// TwinCAT 3 PLC project Untitled1
// ProgramVersion: 3.1.4024.0
// libraries:
//   Tc2_Math, * (Beckhoff Automation GmbH)
//   Tc2_MC2, * (Beckhoff Automation GmbH)
//   Tc2_Standard, * (Beckhoff Automation GmbH)
//   Tc2_System, * (Beckhoff Automation GmbH)
//   Tc2_Utilities, * (Beckhoff Automation GmbH)
//   Tc3_Module, * (Beckhoff Automation GmbH)
//   Tc3_PackML_V2, * (Beckhoff Automation GmbH)
// project tree:
//   DUTs/DUTs/ E_ActWorkUnits.TcDUT (not stored), E_PMLUserUnitMode.TcDUT, E_UnitName.TcDUT (not stored), E_UnitTask.TcDUT (not stored), ST_FeedPara.TcDUT, ST_AxFunctions_1.TcDUT (not stored), ST_AxFunctionsAdmin_.TcDUT, ST_AxFunctionsPTP_1.TcDUT (not stored), ST_ChangeIntoProduction_1.TcDUT, ST_Folder.TcDUT (not stored), ST_FolderCom.TcDUT (not stored), ST_FolderPara.TcDUT, ST_FolderStatus.TcDUT, ST_OneJob.TcDUT (not stored), ST_UnitInfo.TcDUT (not stored)
//   / GlobalTextList.TcGTLO, PlcTask.TcTTO, 视图管理器.TcVMO (not stored)
//   GVLs/ APP_Com.TcDUT, GVL.TcGVL, GVL_Com.TcGVL (not stored), GVL_CONST.TcGVL, GVL_IO.TcGVL
//   POUs/Actuators/ AIN_EL3004.TcPOU (not stored), ANALOG_OUT.TcPOU (not stored), OUTPUT.TcPOU (not stored), SensorikAbblasen.TcPOU
//   POUs/Actuators/Cylinder/ CYLINDER.TcPOU
//   POUs/Actuators/FreqConv/ EcFcCom.TcPOU, IOFcCom.TcPOU
//   POUs/Actuators/Motor/ IOMotor.TcPOU (not stored), IOMotor2Dir.TcPOU (not stored), IOMotorStarDelta.TcPOU
//   POUs/ Axis_PTPV3_CoE.TcPOU, Ax_HMI.TcPOU (not stored), ERROR_HDL.TcPOU (not stored), fbMachine.TcPOU (not stored), FB_Generic.TcPOU (not stored), FB_Visu.TcPOU (not stored), INPUT.TcPOU (not stored), MAIN.TcPOU
//   POUs/EventLogger/ EventStatistik.TcPOU (not stored), EventStatistikData.TcPOU (not stored), EventsWriteToLogbook.TcPOU (not stored)
//   POUs/EventLogger/ReadEvents/ ReadAdsEvents.TcPOU (not stored), READ_ADS_EVENT_DATA.TcDUT, READ_ADS_EVENT_HANDLEINFO.TcDUT (not stored), READ_ADS_EVENT_STREAM.TcDUT, READ_ADS_EVENT_STREAM_DATA_EX.TcDUT (not stored), READ_ADS_EVENT_STREAM_DATA_RAW.TcDUT
//   POUs/EventLogger/TriggerEvents/ EventClass10.TcPOU (not stored), EventClass25.TcPOU, EventClass50.TcPOU (not stored), EventCtrl.TcPOU
//   POUs/Lib/ FB_HydLinearRamp.TcPOU
//   POUs/Lib/EventLogger/TriggerEvents/ EventClass50.TcPOU (not stored), EventCtrl.TcPOU (not stored)
//   POUs/PTP/00_DATATYPE/ AX_JOB.TcPOU (not stored)
//   POUs/PTP/01_Base/ Ax_AdminCtrl.TcPOU (not stored), Ax_HomingCtrl.TcPOU (not stored), Ax_MotionCtrl.TcPOU
//   POUs/PTP/02_Options/Coupling/ Ax_Camming.TcPOU (not stored) (excluded from build), Ax_FlySawCtrl.TcPOU (not stored) (excluded from build), Ax_GearCtrl.TcPOU (not stored)
//   POUs/PTP/02_Options/Drive/ Ax_BrakeCopperIO.TcPOU (not stored)
//   POUs/PTP/02_Options/Drive/CanOpen/ Ax_CanOpenDriveEventCtrl.TcPOU
//   POUs/PTP/02_Options/Drive/Ethercat/ Ax_Ax5000DriveCtrl.TcPOU (not stored), Ax_EcDriveEventCtrl.TcPOU (not stored), Ax_EcMC2DriveCtrl.TcPOU
//   POUs/PTP/02_Options/Drive/Stepper/ Ax_StepperDriveEventCtrl.TcPOU
//   POUs/PTP/02_Options/ErrorNc/ Ax_ErrorNCEventCtrl.TcPOU, Ax_ErrorNCEventMsgCtrl.TcPOU (not stored)
//   POUs/PTP/02_Options/Parameter/ Ax_Para.TcPOU (not stored), AX_PARA_SET_ISTPOS.TcPOU
//   POUs/PTP/02_Options/TouchProbe/ Ax_TouchProbeCtrl.TcPOU
//   POUs/PTP/03_Utilities/ Ax_AutoFctCtrl.TcPOU (not stored), Ax_LoopingDistanceCtrl.TcPOU, Ax_StateUnitCtrl.TcPOU (not stored) (excluded from build), GetAxErrTxt.TcPOU (not stored), MMIN_TO_MMS.TcPOU, MMS_TO_MMIN.TcPOU (not stored), SetOvrVelo.TcPOU
//   POUs/PulseGenerator/ PulseCtrl.TcPOU, PulseGeneratorCtrl.TcPOU
//   POUs/SystemInfo/ SystemInfoCtrl.TcPOU, TaskInfoCtrl.TcPOU
//   POUs/UNIT/fb_Apron/ Analog_To_Angle.TcPOU (not stored), Analog_To_Slide.TcPOU, Angle_To_Analog.TcPOU, fb_Apron.TcPOU (not stored), FB_FoldAbsPos.TcPOU (not stored), FB_SlideAbsPos.TcPOU, Slide_To_Analog.TcPOU
//   POUs/UNIT/fb_BackGauge/ fb_BackGauge.TcPOU (not stored), FB_BGAbsPos.TcPOU, FB_FeedAbsPos.TcPOU (not stored), FB_TblAbsPos.TcPOU (not stored)
//   POUs/UNIT/fb_Clamp/ Anolog_To_Height.TcPOU, fb_Clamp.TcPOU (not stored), FB_ClampJog.TcPOU, FB_ClampLock.TcPOU, FB_ClampMove.TcPOU (not stored), FB_ClampUnlock.TcPOU (not stored), Height_To_Anology.TcPOU (not stored)
//   POUs/UNIT/fb_Slitter/ fb_Slitter.TcPOU (not stored), FB_SlitterAct.TcPOU
//   VISUs/VISUs/Templates/ VIS_TemplateCommand.TcVIS (not stored), VIS_TemplateKeys.TcVIS (not stored), VIS_TemplatePMLStateModel.TcVIS
//   VISUs/VISUs/ VIS_Main.TcVIS (not stored)
// real-time tasks:
//   TASK PlcTask: cycle T#10ms, priority 20, ADS port 350
// motion (NC):
//   TASK NC-Task 1 SAF: cycle T#2ms, priority 4, ADS port 501
//   TASK NC-Task 1 SVB: cycle T#10ms, priority 8, ADS port 511
//   AXIS Axis_T1 (id 1)
//     Dynamic: Acceleration=3740, Deceleration=3740, Jerk=8038.85
//     OtherSettings: AllowMotionCmdToSlave=true
//     encoder EncType=19
//       EncPara: ScaleFactorNumerator=7e-05, MaxCount=#xffffffff, ReferenceSystem=1
//         SoftEndMinControl: Enable=true, Range=-25
//         SoftEndMaxControl: Enable=true, Range=1210
//     drive DrvType=16
//       DrvPara: MaxCount=#xffffffff, DriveControlDWord=#x00020000
//         Analog: VeloReferenz=300, TorqueSetpointScale=10, ScaleFactorActTorque=0.1
//         TimeComp: TaskDelayCycles=1
//     controller CtrType=1
//       CtrPara: PriorControlFactor=1
//         PosDiffControl: Range=10
//         Observer: BandWidth=20
//   AXIS Axis_T2 (id 2)
//     Dynamic: Acceleration=3740, Deceleration=3740, Jerk=8038.85
//     OtherSettings: AllowMotionCmdToSlave=true
//     encoder EncType=19
//       EncPara: ScaleFactorNumerator=7e-05, MaxCount=#xffffffff, ReferenceSystem=1
//         SoftEndMinControl: Enable=true, Range=-25
//         SoftEndMaxControl: Enable=true, Range=1210
//     drive DrvType=16
//       DrvPara: MaxCount=#xffffffff, DriveControlDWord=#x00020000
//         Analog: VeloReferenz=300, TorqueSetpointScale=10, ScaleFactorActTorque=0.1
//         TimeComp: TaskDelayCycles=1
//     controller CtrType=1
//       CtrPara: PriorControlFactor=1
//         PosDiffControl: Range=10
//         Observer: BandWidth=20
//   AXIS Axis_T3 (id 3)
//     Dynamic: Acceleration=3740, Deceleration=3740, Jerk=8038.85
//     OtherSettings: AllowMotionCmdToSlave=true
//     encoder EncType=19
//       EncPara: ScaleFactorNumerator=7e-05, Inverse=true, MaxCount=#xffffffff, ReferenceSystem=1
//         SoftEndMinControl: Range=-25
//         SoftEndMaxControl: Enable=true, Range=1210
//     drive DrvType=16
//       DrvPara: Inverse=true, MaxCount=#xffffffff, DriveControlDWord=#x00020000
//         Analog: VeloReferenz=300, TorqueSetpointScale=10, ScaleFactorActTorque=0.1
//         TimeComp: TaskDelayCycles=1
//     controller CtrType=1
//       CtrPara: PriorControlFactor=1
//         PosDiffControl: Range=10
//         Observer: BandWidth=20
//   AXIS Axis_T4 (id 4)
//     Dynamic: Acceleration=3740, Deceleration=3740, Jerk=8038.85
//     OtherSettings: AllowMotionCmdToSlave=true
//     encoder EncType=19
//       EncPara: ScaleFactorNumerator=7e-05, MaxCount=#xffffffff, ReferenceSystem=1
//         SoftEndMinControl: Enable=true, Range=-25
//         SoftEndMaxControl: Enable=true, Range=1210
//     drive DrvType=16
//       DrvPara: MaxCount=#xffffffff, DriveControlDWord=#x00020000
//         Analog: VeloReferenz=300, TorqueSetpointScale=10, ScaleFactorActTorque=0.1
//         TimeComp: TaskDelayCycles=1
//     controller CtrType=1
//       CtrPara: PriorControlFactor=1
//         PosDiffControl: Range=10
//         Observer: BandWidth=20
//   AXIS Axis_Table (id 9)
//     Dynamic: Acceleration=1200, Deceleration=1200, Jerk=1440
//     PositionAreaControl: Range=200
//     OtherSettings: AllowMotionCmdToSlave=true
//     encoder EncType=19
//       EncPara: Inverse=true, MaxCount=#xffffffff, ReferenceSystem=1
//         SoftEndMinControl: Range=-10
//         SoftEndMaxControl: Enable=true, Range=800
//     drive DrvType=16
//       DrvPara: Inverse=true, MaxCount=#xffffffff, DriveControlDWord=#x00020000
//         Analog: VeloReferenz=300, TorqueSetpointScale=10, ScaleFactorActTorque=0.1
//         TimeComp: TaskDelayCycles=1
//     controller CtrType=1
//       CtrPara: PriorControlFactor=1
//         PosDiffControl: Range=100
//         Observer: BandWidth=20
//   AXIS Axis_Feed (id 5)
//     PositionAreaControl: Range=200
//     OtherSettings: AllowMotionCmdToSlave=true
//     encoder EncType=19
//       EncPara: ScaleFactorNumerator=0.00026, MaxCount=#xffffffff, ReferenceSystem=1
//         SoftEndMinControl: Enable=true, Range=-420
//         SoftEndMaxControl: Enable=true, Range=3900
//     drive DrvType=16
//       DrvPara: MaxCount=#xffffffff, DriveControlDWord=#x00020000
//         Analog: TorqueSetpointScale=10, ScaleFactorActTorque=0.1
//         TimeComp: TaskDelayCycles=1
//     controller CtrType=1
//       CtrPara: PriorControlFactor=1
//         PosDiffControl: Range=200
//         Observer: BandWidth=20
// I/O:
//   DEVICE Device 2 (EtherCAT), AmsNetId 192.168.78.10.3.1
//     Term 24 (EK1100) [EK1100 EtherCAT Coupler (2A E-Bus)]
//       Term 25 (EL1008) [EL1008 8Ch. Dig. Input 24V, 3ms]
//       Term 27 (EL1008) [EL1008 8Ch. Dig. Input 24V, 3ms]
//       Term 28 (EL1008) [EL1008 8Ch. Dig. Input 24V, 3ms]
//       Term 30 (EL1008) [EL1008 8Ch. Dig. Input 24V, 3ms]
//       Term 31 (EL1008) [EL1008 8Ch. Dig. Input 24V, 3ms]
//       Term 33 (EL2008) [EL2008 8Ch. Dig. Output 24V, 0.5A]
//       Term 34 (EL2008) [EL2008 8Ch. Dig. Output 24V, 0.5A]
//       Term 35 (EL2008) [EL2008 8Ch. Dig. Output 24V, 0.5A]
//       Term 36 (EL2008) [EL2008 8Ch. Dig. Output 24V, 0.5A]
//       Term 14 (EL2008) [EL2008 8Ch. Dig. Output 24V, 0.5A]
//       Term 37 (EL3004) [EL3004 4Ch. Ana. Input +/-10V]
//       Term 38 (EL3004) [EL3004 4Ch. Ana. Input +/-10V]
//       Term 39 (EL4004) [EL4004 4Ch. Ana. Output 0-10V, 12bit]
//       Term 41 (EL4024) [EL4024 4Ch. Ana. Output 4-20mA, 12bit]
//       Term 42 (EL4024) [EL4024 4Ch. Ana. Output 4-20mA, 12bit]
//       Term 43 (EL3024) [EL3024 4Ch. Ana. Input 4-20mA DIFF]
//       Term 47 (EL9011) [EL9011 End Terminal]
//     Drive 19 (ASDA-W3-E CoE Drive) [Delta ASDA-W3-E EtherCAT(CoE) Drive]
//       modules: Module 1 (W3 Servo Drive-Axis), Module 2 (W3 Servo Drive-Axis), Module 3 (W3 Servo Drive-Axis), Module 4 (W3 Servo Drive-Axis), Module 5 (W3 Servo Drive-Axis), Module 6 (W3 Servo Drive-Axis)
// variable links:
//   NC-Task 1 SAF/Axes/Axis_Feed <-> Device 2 (EtherCAT)/Drive 19 (ASDA-W3-E CoE Drive)
//     Drive/Inputs/In/nDataIn3[0] <-> Module 6 (W3 Servo Drive-Axis)/1st TxPDO Mapping/Actual Torque
//     Drive/Inputs/In/nDcOutputTime <-> InfoData/DcOutputShift
//     Drive/Inputs/In/nState1 <-> Module 6 (W3 Servo Drive-Axis)/1st TxPDO Mapping/Status Word
//     Drive/Inputs/In/nState2 <-> Module 6 (W3 Servo Drive-Axis)/1st TxPDO Mapping/Status Word @bit 8
//     Drive/Inputs/In/nState4 @bit 1 <-> WcState/InputToggle
//     Drive/Inputs/In/nState4 <-> WcState/WcState
//     Drive/Outputs/Out/nCtrl1 <-> Module 6 (W3 Servo Drive-Axis)/1st RxPDO Mapping/Control Word
//     Drive/Outputs/Out/nCtrl2 <-> Module 6 (W3 Servo Drive-Axis)/1st RxPDO Mapping/Control Word @bit 8
//     Drive/Outputs/Out/nDataOut1 <-> Module 6 (W3 Servo Drive-Axis)/1st RxPDO Mapping/TargetPosition
//     Drive/Outputs/Out/nDataOut2 <-> Module 6 (W3 Servo Drive-Axis)/1st RxPDO Mapping/TargetVelocity
//     Drive/Outputs/Out/nDataOut4[0] <-> Module 6 (W3 Servo Drive-Axis)/1st RxPDO Mapping/Target Torque
//     Enc/Inputs/In/nDataIn1 <-> Module 6 (W3 Servo Drive-Axis)/1st TxPDO Mapping/ActualPosition
//     Enc/Inputs/In/nDataIn3 <-> Module 6 (W3 Servo Drive-Axis)/1st TxPDO Mapping/Touch Probe Pos1 Pos Value
//     Enc/Inputs/In/nDataIn7 <-> Module 6 (W3 Servo Drive-Axis)/1st TxPDO Mapping/ActualVelocity
//     Enc/Inputs/In/nDcInputTime <-> InfoData/DcInputShift
//     Enc/Inputs/In/nState4 @bit 1 <-> WcState/InputToggle
//     Enc/Inputs/In/nState4 <-> WcState/WcState
//     Enc/Inputs/In/nState5 <-> Module 6 (W3 Servo Drive-Axis)/1st TxPDO Mapping/Touch Probe Status
//     Enc/Inputs/In/nState6 <-> Module 6 (W3 Servo Drive-Axis)/1st TxPDO Mapping/Touch Probe Status @bit 8
//     Enc/Outputs/Out/nCtrl5 <-> Module 6 (W3 Servo Drive-Axis)/1st RxPDO Mapping/Touch Probe Function
//     Enc/Outputs/Out/nCtrl6 <-> Module 6 (W3 Servo Drive-Axis)/1st RxPDO Mapping/Touch Probe Function @bit 8
//   NC-Task 1 SAF/Axes/Axis_T1 <-> Device 2 (EtherCAT)/Drive 19 (ASDA-W3-E CoE Drive)
//     Drive/Inputs/In/nDataIn3[0] <-> Module 1 (W3 Servo Drive-Axis)/1st TxPDO Mapping/Actual Torque
//     Drive/Inputs/In/nDcOutputTime <-> InfoData/DcOutputShift
//     Drive/Inputs/In/nState1 <-> Module 1 (W3 Servo Drive-Axis)/1st TxPDO Mapping/Status Word
//     Drive/Inputs/In/nState2 <-> Module 1 (W3 Servo Drive-Axis)/1st TxPDO Mapping/Status Word @bit 8
//     Drive/Inputs/In/nState4 @bit 1 <-> WcState/InputToggle
//     Drive/Inputs/In/nState4 <-> WcState/WcState
//     Drive/Outputs/Out/nCtrl1 <-> Module 1 (W3 Servo Drive-Axis)/1st RxPDO Mapping/Control Word
//     Drive/Outputs/Out/nCtrl2 <-> Module 1 (W3 Servo Drive-Axis)/1st RxPDO Mapping/Control Word @bit 8
//     Drive/Outputs/Out/nDataOut1 <-> Module 1 (W3 Servo Drive-Axis)/1st RxPDO Mapping/TargetPosition
//     Drive/Outputs/Out/nDataOut2 <-> Module 1 (W3 Servo Drive-Axis)/1st RxPDO Mapping/TargetVelocity
//     Drive/Outputs/Out/nDataOut4[0] <-> Module 1 (W3 Servo Drive-Axis)/1st RxPDO Mapping/Target Torque
//     Enc/Inputs/In/nDataIn1 <-> Module 1 (W3 Servo Drive-Axis)/1st TxPDO Mapping/ActualPosition
//     Enc/Inputs/In/nDataIn3 <-> Module 1 (W3 Servo Drive-Axis)/1st TxPDO Mapping/Touch Probe Pos1 Pos Value
//     Enc/Inputs/In/nDataIn7 <-> Module 1 (W3 Servo Drive-Axis)/1st TxPDO Mapping/ActualVelocity
//     Enc/Inputs/In/nDcInputTime <-> InfoData/DcInputShift
//     Enc/Inputs/In/nState4 @bit 1 <-> WcState/InputToggle
//     Enc/Inputs/In/nState4 <-> WcState/WcState
//     Enc/Inputs/In/nState5 <-> Module 1 (W3 Servo Drive-Axis)/1st TxPDO Mapping/Touch Probe Status
//     Enc/Inputs/In/nState6 <-> Module 1 (W3 Servo Drive-Axis)/1st TxPDO Mapping/Touch Probe Status @bit 8
//     Enc/Outputs/Out/nCtrl5 <-> Module 1 (W3 Servo Drive-Axis)/1st RxPDO Mapping/Touch Probe Function
//     Enc/Outputs/Out/nCtrl6 <-> Module 1 (W3 Servo Drive-Axis)/1st RxPDO Mapping/Touch Probe Function @bit 8
//   NC-Task 1 SAF/Axes/Axis_T2 <-> Device 2 (EtherCAT)/Drive 19 (ASDA-W3-E CoE Drive)
//     Drive/Inputs/In/nDataIn3[0] <-> Module 2 (W3 Servo Drive-Axis)/1st TxPDO Mapping/Actual Torque
//     Drive/Inputs/In/nDcOutputTime <-> InfoData/DcOutputShift
//     Drive/Inputs/In/nState1 <-> Module 2 (W3 Servo Drive-Axis)/1st TxPDO Mapping/Status Word
//     Drive/Inputs/In/nState2 <-> Module 2 (W3 Servo Drive-Axis)/1st TxPDO Mapping/Status Word @bit 8
//     Drive/Inputs/In/nState4 @bit 1 <-> WcState/InputToggle
//     Drive/Inputs/In/nState4 <-> WcState/WcState
//     Drive/Outputs/Out/nCtrl1 <-> Module 2 (W3 Servo Drive-Axis)/1st RxPDO Mapping/Control Word
//     Drive/Outputs/Out/nCtrl2 <-> Module 2 (W3 Servo Drive-Axis)/1st RxPDO Mapping/Control Word @bit 8
//     Drive/Outputs/Out/nDataOut1 <-> Module 2 (W3 Servo Drive-Axis)/1st RxPDO Mapping/TargetPosition
//     Drive/Outputs/Out/nDataOut2 <-> Module 2 (W3 Servo Drive-Axis)/1st RxPDO Mapping/TargetVelocity
//     Drive/Outputs/Out/nDataOut4[0] <-> Module 2 (W3 Servo Drive-Axis)/1st RxPDO Mapping/Target Torque
//     Enc/Inputs/In/nDataIn1 <-> Module 2 (W3 Servo Drive-Axis)/1st TxPDO Mapping/ActualPosition
//     Enc/Inputs/In/nDataIn3 <-> Module 2 (W3 Servo Drive-Axis)/1st TxPDO Mapping/Touch Probe Pos1 Pos Value
//     Enc/Inputs/In/nDataIn7 <-> Module 2 (W3 Servo Drive-Axis)/1st TxPDO Mapping/ActualVelocity
//     Enc/Inputs/In/nDcInputTime <-> InfoData/DcInputShift
//     Enc/Inputs/In/nState4 @bit 1 <-> WcState/InputToggle
//     Enc/Inputs/In/nState4 <-> WcState/WcState
//     Enc/Inputs/In/nState5 <-> Module 2 (W3 Servo Drive-Axis)/1st TxPDO Mapping/Touch Probe Status
//     Enc/Inputs/In/nState6 <-> Module 2 (W3 Servo Drive-Axis)/1st TxPDO Mapping/Touch Probe Status @bit 8
//     Enc/Outputs/Out/nCtrl5 <-> Module 2 (W3 Servo Drive-Axis)/1st RxPDO Mapping/Touch Probe Function
//     Enc/Outputs/Out/nCtrl6 <-> Module 2 (W3 Servo Drive-Axis)/1st RxPDO Mapping/Touch Probe Function @bit 8
//   NC-Task 1 SAF/Axes/Axis_T3 <-> Device 2 (EtherCAT)/Drive 19 (ASDA-W3-E CoE Drive)
//     Drive/Inputs/In/nDataIn3[0] <-> Module 3 (W3 Servo Drive-Axis)/1st TxPDO Mapping/Actual Torque
//     Drive/Inputs/In/nDcOutputTime <-> InfoData/DcOutputShift
//     Drive/Inputs/In/nState1 <-> Module 3 (W3 Servo Drive-Axis)/1st TxPDO Mapping/Status Word
//     Drive/Inputs/In/nState2 <-> Module 3 (W3 Servo Drive-Axis)/1st TxPDO Mapping/Status Word @bit 8
//     Drive/Inputs/In/nState4 @bit 1 <-> WcState/InputToggle
//     Drive/Inputs/In/nState4 <-> WcState/WcState
//     Drive/Outputs/Out/nCtrl1 <-> Module 3 (W3 Servo Drive-Axis)/1st RxPDO Mapping/Control Word
//     Drive/Outputs/Out/nCtrl2 <-> Module 3 (W3 Servo Drive-Axis)/1st RxPDO Mapping/Control Word @bit 8
//     Drive/Outputs/Out/nDataOut1 <-> Module 3 (W3 Servo Drive-Axis)/1st RxPDO Mapping/TargetPosition
//     Drive/Outputs/Out/nDataOut2 <-> Module 3 (W3 Servo Drive-Axis)/1st RxPDO Mapping/TargetVelocity
//     Drive/Outputs/Out/nDataOut4[0] <-> Module 3 (W3 Servo Drive-Axis)/1st RxPDO Mapping/Target Torque
//     Enc/Inputs/In/nDataIn1 <-> Module 3 (W3 Servo Drive-Axis)/1st TxPDO Mapping/ActualPosition
//     Enc/Inputs/In/nDataIn3 <-> Module 3 (W3 Servo Drive-Axis)/1st TxPDO Mapping/Touch Probe Pos1 Pos Value
//     Enc/Inputs/In/nDataIn7 <-> Module 3 (W3 Servo Drive-Axis)/1st TxPDO Mapping/ActualVelocity
//     Enc/Inputs/In/nDcInputTime <-> InfoData/DcInputShift
//     Enc/Inputs/In/nState4 @bit 1 <-> WcState/InputToggle
//     Enc/Inputs/In/nState4 <-> WcState/WcState
//     Enc/Inputs/In/nState5 <-> Module 3 (W3 Servo Drive-Axis)/1st TxPDO Mapping/Touch Probe Status
//     Enc/Inputs/In/nState6 <-> Module 3 (W3 Servo Drive-Axis)/1st TxPDO Mapping/Touch Probe Status @bit 8
//     Enc/Outputs/Out/nCtrl5 <-> Module 3 (W3 Servo Drive-Axis)/1st RxPDO Mapping/Touch Probe Function
//     Enc/Outputs/Out/nCtrl6 <-> Module 3 (W3 Servo Drive-Axis)/1st RxPDO Mapping/Touch Probe Function @bit 8
//   NC-Task 1 SAF/Axes/Axis_T4 <-> Device 2 (EtherCAT)/Drive 19 (ASDA-W3-E CoE Drive)
//     Drive/Inputs/In/nDataIn3[0] <-> Module 4 (W3 Servo Drive-Axis)/1st TxPDO Mapping/Actual Torque
//     Drive/Inputs/In/nDcOutputTime <-> InfoData/DcOutputShift
//     Drive/Inputs/In/nState1 <-> Module 4 (W3 Servo Drive-Axis)/1st TxPDO Mapping/Status Word
//     Drive/Inputs/In/nState2 <-> Module 4 (W3 Servo Drive-Axis)/1st TxPDO Mapping/Status Word @bit 8
//     Drive/Inputs/In/nState4 @bit 1 <-> WcState/InputToggle
//     Drive/Inputs/In/nState4 <-> WcState/WcState
//     Drive/Outputs/Out/nCtrl1 <-> Module 4 (W3 Servo Drive-Axis)/1st RxPDO Mapping/Control Word
//     Drive/Outputs/Out/nCtrl2 <-> Module 4 (W3 Servo Drive-Axis)/1st RxPDO Mapping/Control Word @bit 8
//     Drive/Outputs/Out/nDataOut1 <-> Module 4 (W3 Servo Drive-Axis)/1st RxPDO Mapping/TargetPosition
//     Drive/Outputs/Out/nDataOut2 <-> Module 4 (W3 Servo Drive-Axis)/1st RxPDO Mapping/TargetVelocity
//     Drive/Outputs/Out/nDataOut4[0] <-> Module 4 (W3 Servo Drive-Axis)/1st RxPDO Mapping/Target Torque
//     Enc/Inputs/In/nDataIn1 <-> Module 4 (W3 Servo Drive-Axis)/1st TxPDO Mapping/ActualPosition
//     Enc/Inputs/In/nDataIn3 <-> Module 4 (W3 Servo Drive-Axis)/1st TxPDO Mapping/Touch Probe Pos1 Pos Value
//     Enc/Inputs/In/nDataIn7 <-> Module 4 (W3 Servo Drive-Axis)/1st TxPDO Mapping/ActualVelocity
//     Enc/Inputs/In/nDcInputTime <-> InfoData/DcInputShift
//     Enc/Inputs/In/nState4 @bit 1 <-> WcState/InputToggle
//     Enc/Inputs/In/nState4 <-> WcState/WcState
//     Enc/Inputs/In/nState5 <-> Module 4 (W3 Servo Drive-Axis)/1st TxPDO Mapping/Touch Probe Status
//     Enc/Inputs/In/nState6 <-> Module 4 (W3 Servo Drive-Axis)/1st TxPDO Mapping/Touch Probe Status @bit 8
//     Enc/Outputs/Out/nCtrl5 <-> Module 4 (W3 Servo Drive-Axis)/1st RxPDO Mapping/Touch Probe Function
//     Enc/Outputs/Out/nCtrl6 <-> Module 4 (W3 Servo Drive-Axis)/1st RxPDO Mapping/Touch Probe Function @bit 8
//   NC-Task 1 SAF/Axes/Axis_Table <-> Device 2 (EtherCAT)/Drive 19 (ASDA-W3-E CoE Drive)
//     Drive/Inputs/In/nDataIn3[0] <-> Module 5 (W3 Servo Drive-Axis)/1st TxPDO Mapping/Actual Torque
//     Drive/Inputs/In/nDcOutputTime <-> InfoData/DcOutputShift
//     Drive/Inputs/In/nState1 <-> Module 5 (W3 Servo Drive-Axis)/1st TxPDO Mapping/Status Word
//     Drive/Inputs/In/nState2 <-> Module 5 (W3 Servo Drive-Axis)/1st TxPDO Mapping/Status Word @bit 8
//     Drive/Inputs/In/nState4 @bit 1 <-> WcState/InputToggle
//     Drive/Inputs/In/nState4 <-> WcState/WcState
//     Drive/Outputs/Out/nCtrl1 <-> Module 5 (W3 Servo Drive-Axis)/1st RxPDO Mapping/Control Word
//     Drive/Outputs/Out/nCtrl2 <-> Module 5 (W3 Servo Drive-Axis)/1st RxPDO Mapping/Control Word @bit 8
//     Drive/Outputs/Out/nDataOut1 <-> Module 5 (W3 Servo Drive-Axis)/1st RxPDO Mapping/TargetPosition
//     Drive/Outputs/Out/nDataOut2 <-> Module 5 (W3 Servo Drive-Axis)/1st RxPDO Mapping/TargetVelocity
//     Drive/Outputs/Out/nDataOut4[0] <-> Module 5 (W3 Servo Drive-Axis)/1st RxPDO Mapping/Target Torque
//     Enc/Inputs/In/nDataIn1 <-> Module 5 (W3 Servo Drive-Axis)/1st TxPDO Mapping/ActualPosition
//     Enc/Inputs/In/nDataIn3 <-> Module 5 (W3 Servo Drive-Axis)/1st TxPDO Mapping/Touch Probe Pos1 Pos Value
//     Enc/Inputs/In/nDataIn7 <-> Module 5 (W3 Servo Drive-Axis)/1st TxPDO Mapping/ActualVelocity
//     Enc/Inputs/In/nDcInputTime <-> InfoData/DcInputShift
//     Enc/Inputs/In/nState4 @bit 1 <-> WcState/InputToggle
//     Enc/Inputs/In/nState4 <-> WcState/WcState
//     Enc/Inputs/In/nState5 <-> Module 5 (W3 Servo Drive-Axis)/1st TxPDO Mapping/Touch Probe Status
//     Enc/Inputs/In/nState6 <-> Module 5 (W3 Servo Drive-Axis)/1st TxPDO Mapping/Touch Probe Status @bit 8
//     Enc/Outputs/Out/nCtrl5 <-> Module 5 (W3 Servo Drive-Axis)/1st RxPDO Mapping/Touch Probe Function
//     Enc/Outputs/Out/nCtrl6 <-> Module 5 (W3 Servo Drive-Axis)/1st RxPDO Mapping/Touch Probe Function @bit 8
//   Untitled1/Untitled1 Instance <-> Device 2 (EtherCAT)/Term 24 (EK1100)/Term 14 (EL2008)
//     PlcTask Outputs/GVL_IO.Out_EMG_RopeStop <-> Channel 8/Output
//     PlcTask Outputs/GVL_IO.Out_FlipCupSuction1 <-> Channel 2/Output
//     PlcTask Outputs/GVL_IO.Out_FlipCupSuction2 <-> Channel 4/Output
//     PlcTask Outputs/GVL_IO.Out_FlipCupVent1 <-> Channel 1/Output
//     PlcTask Outputs/GVL_IO.Out_FlipCupVent2 <-> Channel 3/Output
//     PlcTask Outputs/GVL_IO.Out_bak54 <-> Channel 5/Output
//     PlcTask Outputs/GVL_IO.Out_bak55 <-> Channel 6/Output
//     PlcTask Outputs/GVL_IO.Out_bak56 <-> Channel 7/Output
//   Untitled1/Untitled1 Instance <-> Device 2 (EtherCAT)/Term 24 (EK1100)/Term 25 (EL1008)
//     PlcTask Inputs/GVL_IO.In_btnReset <-> Channel 8/Input
//     PlcTask Inputs/GVL_IO.In_pedal1_Clamp <-> Channel 2/Input
//     PlcTask Inputs/GVL_IO.In_pedal1_Fold <-> Channel 5/Input
//     PlcTask Inputs/GVL_IO.In_pedal1_Gripper <-> Channel 6/Input
//     PlcTask Inputs/GVL_IO.In_pedal1_Slitter <-> Channel 3/Input
//     PlcTask Inputs/GVL_IO.In_pedal1_SlitterBack <-> Channel 4/Input
//     PlcTask Inputs/GVL_IO.In_pedal1_UnClamp <-> Channel 1/Input
//     PlcTask Inputs/GVL_IO.In_swOperator <-> Channel 7/Input
//   Untitled1/Untitled1 Instance <-> Device 2 (EtherCAT)/Term 24 (EK1100)/Term 27 (EL1008)
//     PlcTask Inputs/GVL_IO.In_sigBtmApron_FoldHome <-> Channel 7/Input
//     PlcTask Inputs/GVL_IO.In_sigBtmApron_SlideFWD <-> Channel 8/Input
//     PlcTask Inputs/GVL_IO.In_sigSlitLmt0 <-> Channel 1/Input
//     PlcTask Inputs/GVL_IO.In_sigSlitLmt1 <-> Channel 3/Input
//     PlcTask Inputs/GVL_IO.In_sigSlitSlw0 <-> Channel 2/Input
//     PlcTask Inputs/GVL_IO.In_sigSlitSlw1 <-> Channel 4/Input
//     PlcTask Inputs/GVL_IO.In_sigTopApron_FoldHome <-> Channel 5/Input
//     PlcTask Inputs/GVL_IO.In_sigTopApron_SlideFWD <-> Channel 6/Input
//   Untitled1/Untitled1 Instance <-> Device 2 (EtherCAT)/Term 24 (EK1100)/Term 28 (EL1008)
//     PlcTask Inputs/GVL_IO.In_SigSheetDetect1 <-> Channel 7/Input
//     PlcTask Inputs/GVL_IO.In_SigSheetDetect2 <-> Channel 8/Input
//     PlcTask Inputs/GVL_IO.In_bak35 <-> Channel 6/Input
//     PlcTask Inputs/GVL_IO.In_sigBoardPresent <-> Channel 5/Input
//     PlcTask Inputs/GVL_IO.In_sigClampMute <-> Channel 1/Input
//     PlcTask Inputs/GVL_IO.In_sigGaugingFrnt <-> Channel 2/Input
//     PlcTask Inputs/GVL_IO.In_sigGaugingMid <-> Channel 3/Input
//     PlcTask Inputs/GVL_IO.In_sigGaugingRear <-> Channel 4/Input
//   Untitled1/Untitled1 Instance <-> Device 2 (EtherCAT)/Term 24 (EK1100)/Term 30 (EL1008)
//     PlcTask Inputs/GVL_IO.In_EMG_RopeStop <-> Channel 6/Input
//     PlcTask Inputs/GVL_IO.In_sigLC_H <-> Channel 5/Input
//     PlcTask Inputs/GVL_IO.In_sigLC_VLong <-> Channel 4/Input
//     PlcTask Inputs/GVL_IO.In_sigLC_VShort <-> Channel 3/Input
//     PlcTask Inputs/GVL_IO.In_sigLaserFinger <-> Channel 2/Input
//     PlcTask Inputs/GVL_IO.In_sigLubeJam <-> Channel 8/Input
//     PlcTask Inputs/GVL_IO.In_sigPumpJam <-> Channel 7/Input
//     PlcTask Inputs/GVL_IO.In_swLC_Enable <-> Channel 1/Input
//   Untitled1/Untitled1 Instance <-> Device 2 (EtherCAT)/Term 24 (EK1100)/Term 31 (EL1008)
//     PlcTask Inputs/GVL_IO.In_EMG_HandleCabinet <-> Channel 2/Input
//     PlcTask Inputs/GVL_IO.In_EMG_MainCabinet <-> Channel 1/Input
//     PlcTask Inputs/GVL_IO.In_PowerON <-> Channel 3/Input
//     PlcTask Inputs/GVL_IO.In_PumpLow_Alarm <-> Channel 7/Input
//     PlcTask Inputs/GVL_IO.In_VltA_Running <-> Channel 4/Input
//     PlcTask Inputs/GVL_IO.In_VltB_Running <-> Channel 5/Input
//     PlcTask Inputs/GVL_IO.In_VltSlitter_Running <-> Channel 8/Input
//     PlcTask Inputs/GVL_IO.In_Vlt_Alarm <-> Channel 6/Input
//   Untitled1/Untitled1 Instance <-> Device 2 (EtherCAT)/Term 24 (EK1100)/Term 33 (EL2008)
//     PlcTask Outputs/GVL_IO.Out_ClampDown <-> Channel 2/Output
//     PlcTask Outputs/GVL_IO.Out_ClampUp <-> Channel 1/Output
//     PlcTask Outputs/GVL_IO.Out_PumpA_Load_Heav <-> Channel 6/Output
//     PlcTask Outputs/GVL_IO.Out_PumpA_Load_Ligh <-> Channel 5/Output
//     PlcTask Outputs/GVL_IO.Out_PumpB_Load_Heav <-> Channel 8/Output
//     PlcTask Outputs/GVL_IO.Out_PumpB_Load_Ligh <-> Channel 7/Output
//     PlcTask Outputs/GVL_IO.Out_SuctionCup1Suction <-> Channel 4/Output
//     PlcTask Outputs/GVL_IO.Out_SuctionCup1Vent <-> Channel 3/Output
//   Untitled1/Untitled1 Instance <-> Device 2 (EtherCAT)/Term 24 (EK1100)/Term 34 (EL2008)
//     PlcTask Outputs/GVL_IO.Out_GaugingF_Ext <-> Channel 1/Output
//     PlcTask Outputs/GVL_IO.Out_GaugingF_Rtn <-> Channel 2/Output
//     PlcTask Outputs/GVL_IO.Out_GaugingR_Ext <-> Channel 3/Output
//     PlcTask Outputs/GVL_IO.Out_GaugingR_Rtn <-> Channel 4/Output
//     PlcTask Outputs/GVL_IO.Out_Gripper <-> Channel 5/Output
//     PlcTask Outputs/GVL_IO.Out_Gripper2 <-> Channel 6/Output
//     PlcTask Outputs/GVL_IO.Out_GripperDatum_S0 <-> Channel 7/Output
//     PlcTask Outputs/GVL_IO.Out_GripperDatum_S1 <-> Channel 8/Output
//   Untitled1/Untitled1 Instance <-> Device 2 (EtherCAT)/Term 24 (EK1100)/Term 35 (EL2008)
//     PlcTask Outputs/GVL_IO.Out_LubePump <-> Channel 6/Output
//     PlcTask Outputs/GVL_IO.Out_PumpA_ST <-> Channel 1/Output
//     PlcTask Outputs/GVL_IO.Out_PumpB_ST <-> Channel 2/Output
//     PlcTask Outputs/GVL_IO.Out_SlitterBwd <-> Channel 4/Output
//     PlcTask Outputs/GVL_IO.Out_SlitterFwd <-> Channel 3/Output
//     PlcTask Outputs/GVL_IO.Out_SlitterSpeed <-> Channel 5/Output
//     PlcTask Outputs/GVL_IO.Out_SuctionCup2Suction <-> Channel 8/Output
//     PlcTask Outputs/GVL_IO.Out_SuctionCup2Vent <-> Channel 7/Output
//   Untitled1/Untitled1 Instance <-> Device 2 (EtherCAT)/Term 24 (EK1100)/Term 36 (EL2008)
//     PlcTask Outputs/GVL_IO.Out_Gripper3 <-> Channel 8/Output
//     PlcTask Outputs/GVL_IO.Out_Led_Green <-> Channel 7/Output
//     PlcTask Outputs/GVL_IO.Out_Led_Red <-> Channel 5/Output
//     PlcTask Outputs/GVL_IO.Out_Led_Yellow <-> Channel 6/Output
//     PlcTask Outputs/GVL_IO.Out_OpLed_Beep <-> Channel 4/Output
//     PlcTask Outputs/GVL_IO.Out_OpLed_Green <-> Channel 3/Output
//     PlcTask Outputs/GVL_IO.Out_OpLed_Red <-> Channel 1/Output
//     PlcTask Outputs/GVL_IO.Out_OpLed_Yellow <-> Channel 2/Output
//   Untitled1/Untitled1 Instance <-> Device 2 (EtherCAT)/Term 24 (EK1100)/Term 37 (EL3004)
//     PlcTask Inputs/GVL_IO.ANALOG_in_BtmApronFold <-> AI Standard Channel 3/Value
//     PlcTask Inputs/GVL_IO.ANALOG_in_BtmApronSlide <-> AI Standard Channel 4/Value
//     PlcTask Inputs/GVL_IO.ANALOG_in_TopApronFold <-> AI Standard Channel 1/Value
//     PlcTask Inputs/GVL_IO.ANALOG_in_TopApronSlide <-> AI Standard Channel 2/Value
//   Untitled1/Untitled1 Instance <-> Device 2 (EtherCAT)/Term 24 (EK1100)/Term 38 (EL3004)
//     PlcTask Inputs/GVL_IO.ANALOG_in_ClampHeight <-> AI Standard Channel 1/Value
//     PlcTask Inputs/GVL_IO.ANALOG_in_PumpPress <-> AI Standard Channel 2/Value
//     PlcTask Inputs/GVL_IO.ANALOG_in_bak23 <-> AI Standard Channel 3/Value
//     PlcTask Inputs/GVL_IO.ANALOG_in_bak24 <-> AI Standard Channel 4/Value
//   Untitled1/Untitled1 Instance <-> Device 2 (EtherCAT)/Term 24 (EK1100)/Term 39 (EL4004)
//     PlcTask Outputs/GVL_IO.ANALOG_out_PumpA <-> AO Outputs Channel 1/Analog output
//     PlcTask Outputs/GVL_IO.ANALOG_out_PumpB <-> AO Outputs Channel 2/Analog output
//     PlcTask Outputs/GVL_IO.ANALOG_out_bak3 <-> AO Outputs Channel 3/Analog output
//     PlcTask Outputs/GVL_IO.ANALOG_out_bak4 <-> AO Outputs Channel 4/Analog output
//   Untitled1/Untitled1 Instance <-> Device 2 (EtherCAT)/Term 24 (EK1100)/Term 41 (EL4024)
//     PlcTask Outputs/GVL_IO.ANALOG_out_BtmApronFold <-> AO Outputs Channel 1/Analog output
//     PlcTask Outputs/GVL_IO.ANALOG_out_BtmApronSlide <-> AO Outputs Channel 2/Analog output
//   Untitled1/Untitled1 Instance <-> Device 2 (EtherCAT)/Term 24 (EK1100)/Term 42 (EL4024)
//     PlcTask Outputs/GVL_IO.ANALOG_out_ClampDown <-> AO Outputs Channel 1/Analog output
//     PlcTask Outputs/GVL_IO.ANALOG_out_ClampUp <-> AO Outputs Channel 2/Analog output
//     PlcTask Outputs/GVL_IO.ANALOG_out_TopApronFold <-> AO Outputs Channel 3/Analog output
//     PlcTask Outputs/GVL_IO.ANALOG_out_TopApronSlide <-> AO Outputs Channel 4/Analog output
//   Untitled1/Untitled1 Instance <-> Device 2 (EtherCAT)/Term 24 (EK1100)/Term 43 (EL3024)
//     PlcTask Inputs/GVL_IO.ANALOG_in_LiquidHeight <-> AI Standard Channel 2/Value
//     PlcTask Inputs/GVL_IO.ANALOG_in_PumpTemp <-> AI Standard Channel 1/Value
//     PlcTask Inputs/GVL_IO.ANALOG_in_bak43 <-> AI Standard Channel 3/Value
//     PlcTask Inputs/GVL_IO.ANALOG_in_bak44 <-> AI Standard Channel 4/Value
//   Untitled1/Untitled1 Instance <-> NC-Task 1 SAF/Axes/Axis_Feed
//     PlcTask Inputs/MAIN.fbMachine.fbBackGauge.Axis_Feed.ref.NcToPlc <-> Outputs/ToPlc
//     PlcTask Outputs/MAIN.fbMachine.fbBackGauge.Axis_Feed.ref.PlcToNc <-> Inputs/FromPlc
//   Untitled1/Untitled1 Instance <-> NC-Task 1 SAF/Axes/Axis_T1
//     PlcTask Inputs/MAIN.fbMachine.fbBackGauge.Axis_T1.ref.NcToPlc <-> Outputs/ToPlc
//     PlcTask Outputs/MAIN.fbMachine.fbBackGauge.Axis_T1.ref.PlcToNc <-> Inputs/FromPlc
//   Untitled1/Untitled1 Instance <-> NC-Task 1 SAF/Axes/Axis_T2
//     PlcTask Inputs/MAIN.fbMachine.fbBackGauge.Axis_T2.ref.NcToPlc <-> Outputs/ToPlc
//     PlcTask Outputs/MAIN.fbMachine.fbBackGauge.Axis_T2.ref.PlcToNc <-> Inputs/FromPlc
//   Untitled1/Untitled1 Instance <-> NC-Task 1 SAF/Axes/Axis_T3
//     PlcTask Inputs/MAIN.fbMachine.fbBackGauge.Axis_T3.ref.NcToPlc <-> Outputs/ToPlc
//     PlcTask Outputs/MAIN.fbMachine.fbBackGauge.Axis_T3.ref.PlcToNc <-> Inputs/FromPlc
//   Untitled1/Untitled1 Instance <-> NC-Task 1 SAF/Axes/Axis_T4
//     PlcTask Inputs/MAIN.fbMachine.fbBackGauge.Axis_T4.ref.NcToPlc <-> Outputs/ToPlc
//     PlcTask Outputs/MAIN.fbMachine.fbBackGauge.Axis_T4.ref.PlcToNc <-> Inputs/FromPlc
//   Untitled1/Untitled1 Instance <-> NC-Task 1 SAF/Axes/Axis_Table
//     PlcTask Inputs/MAIN.fbMachine.fbBackGauge.Axis_Table.ref.NcToPlc <-> Outputs/ToPlc
//     PlcTask Outputs/MAIN.fbMachine.fbBackGauge.Axis_Table.ref.PlcToNc <-> Inputs/FromPlc

CONFIGURATION Untitled1
    RESOURCE PLC ON TwinCAT3
        TASK PlcTask(INTERVAL := T#10ms, PRIORITY := 20);
        PROGRAM MAIN WITH PlcTask : MAIN;
    END_RESOURCE
END_CONFIGURATION

// ---- DUTs/DUTs/E_PMLUserUnitMode.TcDUT
//Enumeration for User Modes
TYPE E_PMLUserUnitMode : (
	ePMLUnitMode_SemiAuto		:=  4,
	ePMLUnitMode_AutoSlitter	:=  5,
	ePMLUnitMode_Auto			:=  6,
	ePMLUnitMode_AutoFeed		:=  7,
	ePMLUnitMode_Usermode6 		:=  9,
	ePMLUnitMode_Usermode5 		:=  8,
	ePMLUnitMode_Usermode7 		:=  10
) DINT;
END_TYPE

// ---- DUTs/DUTs/ST_FeedPara.TcDUT
TYPE ST_FeedPara :
STRUCT
	Width:UINT;
	Length:UINT;
	Thickness:REAL;
	Quantity :UINT;
	Groups:UINT;
	Total:UINT;
	
	FeedPOS1:REAL;
	FeedPOS2:REAL;
	
END_STRUCT
END_TYPE

// ---- DUTs/DUTs/ST_AxFunctionsAdmin_.TcDUT
//structure includes axisfunctions
TYPE ST_AxFunctionsAdmin_ :
STRUCT
	Power	: MC_Power;
	Reset	: MC_Reset;
END_STRUCT
END_TYPE

// ---- DUTs/DUTs/ST_ChangeIntoProduction_1.TcDUT
//structure for a visu userwindow, to chnage into productionmode
TYPE ST_ChangeIntoProduction_1 :
STRUCT
	bYes		: BOOL;
	bNo			: BOOL;
	bYesReset	: BOOL;
END_STRUCT
END_TYPE

// ---- DUTs/DUTs/ST_FolderPara.TcDUT
TYPE ST_FolderPara :
STRUCT
	//[GlobalSwitch]
	swLightHeavy,swSimplexDuplex	:BOOL;
	swSlitterVelocity,swLoadingTable,swAngleDisplay	:BOOL;
	swLightCurtainEn	:BOOL;
	swClampOpen_InManual,swClampOpen_InAuto	:BOOL;
	swFeedMechanism:BOOL;
	// [ClampHeight]
	Clamp_LowPos,Clamp_MidPos,Clamp_HighPos	:REAL;
	Clamp_MaxPos,ClampHalfPos	:REAL;
	Clamp_PressFlat,Clamp_FoldEnd	:REAL;
	Clamp_FeedPos:REAL;
	// [BackgaugeApron]
	BackgaugeMaxPos,BackgaugeMinPos		:REAL;
	SlitterOffset	:REAL;			(*钳口－切刀的距离*)
	BtmApronZeroPosition,TopApronZeroPosition	:REAL;
	SquashBackstop_Top,SquashBackstop_Btm,SquashBackstop_External	:REAL;
	SquashBackstop_OpenTop,SquashBackstop_OpenBtm	:REAL;
	MT1_BackstopZero	:REAL;
	MT2_BackstopZero,MT3_BackstopZero,MT4_BackstopZero	:REAL;
	Flip_TableToClampDistance	:REAL;
	Flip_SuctionCupInstallPos	:REAL;
	Flip_PickupClampHeight		:REAL;
	Flip_TopApronPickupAngle	:REAL;
	Flip_TablePickupOffset		:REAL;
	//[ManualOldSelect]
	FoldMode,PosDatumPoint	:BOOL;
	SetFoldAngle,SetMoveBackgauge,SetTopApronSlide,SetBtmApronSlide,SetLoadingTable	:REAL;
	AngleAdditSel_id 		:REAL;

	
	bSemiAuto_Step,bSemiAuto_Slitter,bSemiAuto_BackGauge	:BOOL;
	//	[FEED]
	FeedOffset,FeedPosition	:REAL;
	SetMoveFeed	:REAL;
	
	BackGauge_MaxPos,	BackGauge_MinPos	:REAL;
	
	TopAngleAddit,BtmAngleAddit		:ARRAY[0..14] OF REAL;

END_STRUCT
END_TYPE

// ---- DUTs/DUTs/ST_FolderStatus.TcDUT
TYPE ST_FolderStatus :
STRUCT
	Mode	:INT;
	Operator	:INT;
	FoldRunning	:BOOL;
	Gripper,Gripper2	:BOOL;
	GripperClose,GripperHalf,GripperOpen :BOOL;

	SuctionCup1,SuctionCup2	:BOOL;	//真空吸盘
	FlipSuctionCup			:BOOL;	//翻转真空吸盘
	
	Slitter_AtHome	:BOOL;
	SlitterAtSlow	:BOOL;
	
	BackGauge_AtHome	:BOOL;
	BG_Coupled	:BOOL;
	
	ApronTopSlide_AtWork,ApronTopSlide_AtMax	:BOOL;
	ApronBtmSlide_AtWork,ApronBtmSlide_AtMax	:BOOL;
	ApronTopSlide_AtSlow,ApronBtmSlide_AtSlow	:BOOL;
	
	ApronTopFold_AtHome,ApronTopFold_AtMax		:BOOL;
	ApronBtmFold_AtHome,ApronBtmFold_AtMax		:BOOL;
	ApronFold_AtSlow	:BOOL;
	
	Clamp_AtPressPoint	:BOOL;
	Clamp_AtZeroPoint	:BOOL;
	Clamp_LtHalfPoint	:BOOL;
	Clamp_GtLowPoint	:BOOL;
	Clamp_Slow			:BOOL;
	
	Table_AtHome	:BOOL;
	
	Feed_AtHome	:BOOL;
	Feed_AtWork	:BOOL;
	
	Flip_WorkDone :BOOL;
	Flip_AtWork :BOOL;
END_STRUCT
END_TYPE

// ---- GVLs/APP_Com.TcDUT
TYPE APP_Com :
STRUCT
	bBackStationPosFinish:BOOL;
	bBendStationPosFinish:BOOL;
END_STRUCT
END_TYPE

// ---- POUs/EventLogger/ReadEvents/READ_ADS_EVENT_DATA.TcDUT
TYPE READ_ADS_EVENT_DATA :
STRUCT
	Class			: E_TcEventClass;
	id				: DWORD;
	State			: DWORD;
	Question		: DWORD;
	SourceId		: DWORD;
	Source			: STRING(80);
	DateAndTime		: DT;
	Computer		: STRING(80);
	MsgText			: STRING(500);
END_STRUCT
END_TYPE

// ---- POUs/EventLogger/ReadEvents/READ_ADS_EVENT_STREAM.TcDUT
TYPE READ_ADS_EVENT_STREAM :
STRUCT
	cbStream		: DWORD; 			(* size OF this structure, including all following TcGetEventParams structures *)
	count			: DWORD;
	data			: READ_ADS_EVENT_STREAM_DATA_RAW;	(* Stream OF TcGetEventParams *)
END_STRUCT
END_TYPE

// ---- POUs/EventLogger/ReadEvents/READ_ADS_EVENT_STREAM_DATA_RAW.TcDUT
TYPE READ_ADS_EVENT_STREAM_DATA_RAW :
STRUCT
	cb						: DWORD;
	InvokeId				: DWORD;
	Id						: DWORD;
	SrcId					: DWORD;
	addr					: ARRAY [1..8] OF BYTE;
	Class					: DWORD;
	Flags					: DWORD;
	Prio					: DWORD;
	State					: DWORD;
	UserData				: DWORD;
	zFmtProgId				: STRING(31);

	TimeSignaled			: T_FILETIME;
	TimeReset				: T_FILETIME;
	TimeConfirm				: T_FILETIME;

	evtData					: READ_ADS_EVENT_STREAM_DATA_EX;
	
END_STRUCT
END_TYPE

// ---- GVLs/GVL.TcGVL
VAR_GLOBAL
		PackTags					: ST_PackMLv30;					//PackTags
// Dekl. Global Taktmerker
	pulse													: PulseCtrl;

	// Dekl. GetSystemInfo
	SysInfo													: SystemInfoCtrl;
	
		bButtonProductionReq		: BOOL;							//TRUE when a mode change to PRODUCTION is requested
		
		
		aUnitInfo					: ARRAY [1..12] OF ST_UnitInfo;	//Array includes the states and modes of machineunits	
		aCaption					: ARRAY [1..12] OF STRING := ['F1','F2','F3','F4','F5','F6','F7','F8','F9','F10','F11','F12'];
		aKeyPressed					: ARRAY [1..12] OF BOOL;	
		
		//Axis1:AXIS_REF;
		
		SemiAuto_ActJob	:ST_OneJob;
		SemiAuto_LastJob , SemiAuto_NextJob	:ST_OneJob;
		SlitterAuto_ActJob_Width	:REAL;
		SlitterAuto_ActJob_Num	:REAL;
		FeedAuto_Job:ST_FeedPara;
		
	FirstDualPump_5m	:BOOL;
	
	bReset	:BOOL;
	rtReset	:R_TRIG;
	pedal_UnClamp,	pedal_Clamp		:BOOL;
	pedal_Slitter,	pedal_SlitterBack	:BOOL;
	pedal_Fold,	pedal_Gripper	:BOOL;

	
	Hmi_bArray		AT%MB0:ARRAY[0..299] OF BOOL;
	Hmi_iArray		AT%MW300:ARRAY[0..299] OF UINT;
	Hmi_rArray		AT%MD1000:ARRAY[0..299] OF REAL;
	
	
	
	Hmi_iSemiAuto 	AT%MW8000:ARRAY[0..299] OF INT;
	Hmi_iAuto 		AT%MW3000:ARRAY[0..299] OF INT;
	Hmi_rSlitter	AT%MW4000:ARRAY[0..29] OF REAL;
	
	
		
	stFolder		:ST_FOLDER;
	
	
	
	b_sigLC_VShort: BOOL;
	gvl_rtEnSemiAuto: R_trig;
	gvl_rtEnSlitter: R_trig;
	
	gvl_bSlipPatch_BtmSlide,gvl_bSlipPatch_BtmFold		:BOOL;

	
END_VAR



VAR_GLOBAL PERSISTENT
	i12345	:INT;
	b_SafeSysEn: BOOL;
	
	Operators	:UINT;
	LubePumpCount	:INT;
	
	stFolderPara	:ST_FolderPara;
	AngleMap_Top	AT%MW5000	:ARRAY[0..199] OF INT;
	AngleMap_Btm	AT%MW5500	:ARRAY[0..199] OF INT;
	HeightMap		AT%MW6000	:ARRAY[0..399] OF INT;
	AdvPara			AT%MW9000	:ARRAY[0..99]  OF REAL;
END_VAR


VAR_GLOBAL RETAIN
	gvl_rtEnManual: R_trig;
END_VAR

// ---- GVLs/GVL_CONST.TcGVL
VAR_GLOBAL CONSTANT
	PUMP_FREQ_IDLE: USINT  :=143;
	
	
	CONST_APRON_SLIDE_DECWINDOW			:REAL	:=30.0;				(*台板滑动减速距离*)
	CONST_APRON_SLIDE_WINDOW			:REAL	:=5.0;				(*台板滑动定位窗口*)
	CONST_APRON_TOPSLIDE_POS0		:REAL	:=0.0;			(*AtWork时为0*)
	CONST_APRON_TOPSLIDE_POS1		:REAL	:=50.0;
	CONST_APRON_TOPSLIDE_POS2		:REAL	:=100.0;
	CONST_APRON_TOPSLIDE_POS3		:REAL	:=195.0;		(*退回时为200*)

	CONST_APRON_BTMSLIDE_POS0		:REAL	:=0.0;			(*AtWork时为0*)
	CONST_APRON_BTMSLIDE_POS1		:REAL	:=50.0;
	CONST_APRON_BTMSLIDE_POS2		:REAL	:=100.0;
	CONST_APRON_BTMSLIDE_POS3		:REAL	:=195.0;		(*退回时为200*)

	
	CONST_APRON_FOLD_DECWINDOW			:REAL	:=10.0;				(*台板折弯减速距离*)
	CONST_APRON_FOLD_WINDOW				:REAL	:=20.0;				(*台板折弯定位窗口*)
	CONST_APRON_TOPFOLD_POS_MAX			:REAL	:=200.0;
	CONST_APRON_TOPFOLD_POS_MIN			:REAL	:=0.0;
	CONST_APRON_BTMFOLD_POS_Max			:REAL	:=200.0;
	CONST_APRON_BTMFOLD_POS_MIN			:REAL	:=0.0;
	CONST_APRON_TOPFOLD_LIMIT			:REAL	:=150.0;		(*上翻板折弯 -- 机械极限*)
	CONST_APRON_BTMFOLD_LIMIT			:REAL	:=150.0;		(*下翻板折弯 -- 机械极限*)
	
	CONST_CLAMP_LIGHT_PRESSURE_SETPOINT	:REAL	:=7.0;		(*钳口压紧的压力值*)	
	CONST_CLAMP_HEAVY_PRESSURE_SETPOINT	:INT	:=100;
	CONST_CLAMP_POS_CALIBRATION	:INT	:=4;		(*CLAMP calibration 定义为认为闭合的位置*)
	CONST_CLAMP_POS_HALF	:INT	:=45;
	CONST_CLAMP_POS_LOW	:INT	:=3;
	CONST_CLAMP_SPEED_CREEP	:INT	:=500;
	CONST_CLAMP_SPEED_HIGH	:INT	:=4000;
	CONST_CLAMP_MAXCONVERT		:DINT	:=10000;			(*模拟量为32767时对应的值*)
	
	CONST_BACKGAUGE_SPEED_HIGH	:INT	:=200;
	CONST_BACKGAUGE_SPEED_LOW	:INT	:=50;
	CONST_BACKGAUGE_SPEED_CREEP	:INT	:=20;
	CONST_BACKGAUGE_POS_ZERO	:INT	:=0;
	CONST_BACKGAUGE_POS_NegPlus	:INT	:=-20;
	CONST_BACKGAUGE_POS_Window	:REAL	:=2.0;
	
	CONST_BACKGAUGE_ATTACH_PUSH		:REAL	:=0.0;		(*附加量-PUSH*)
	CONST_BACKGAUGE_ATTACH_GRIP		:REAL	:=10.0;		(*附加量-GRIP*)
	CONST_BACKGAUGE_ATTACH_OVERGRIP	:REAL	:=30.0;		(*附加量-OVERGRIP*)
	CONST_BACKGAUGE_ATTACH_BACK		:REAL	:=60.0;		(*附加量-BACK*)
	
	CONST_TABLE_SPEED_HIGH	:INT	:=300;
	CONST_TABLE_POS_MAX		:INT	:=800;
	CONST_TABLE_POS_MIN		:INT	:=0;
	
	CONST_FEED_SPEED_HIGH	:INT	:=800;
	CONST_FEED_SPEED_LOW	:INT	:=500;
	CONST_FEED_SPEED_CREEP	:INT	:=20;
	CONST_FEED_POS_ZERO	:INT	:=0;
	CONST_FEED_POS_NegPlus	:INT	:=-20;
	CONST_FEED_POS_Window	:REAL	:=2.0;
	CONST_FEED_POS_MAX		:INT	:=3900;
	CONST_FEED_POS_MIN		:INT	:=-450;
	
END_VAR

VAR_GLOBAL 
	CNST_HYD_IDLE_SPD					:REAL	:=0.0;	//	油泵待机速度
	CNST_HYD_PUMP_ACC_STEP				:REAL	:=40.0;	//	油泵斜坡加速步长_初始值
	CNST_HYD_PUMP_DEC_STEP				:REAL	:=60.0;	//	油泵斜坡减速步长_初始值
	CNST_HYD_APRON_SLIDE_ACC_STEP		:REAL	:=80.0;	//	翻板滑动比例阀加速步长_初始值
	CNST_HYD_APRON_SLIDE_DEC_STEP		:REAL	:=120.0;	//	翻板滑动比例阀减速步长_初始值
	CNST_HYD_APRON_SLIDE_MIN_OUTPUT		:REAL	:=220.0;	//	翻板滑动比例阀最小起跳量_初始值
	CNST_HYD_APRON_FOLD_ACC_STEP		:REAL	:=70.0;	//	翻板折弯比例阀加速步长_初始值
	CNST_HYD_APRON_FOLD_DEC_STEP		:REAL	:=110.0;	//	翻板折弯比例阀减速步长_初始值
	CNST_HYD_APRON_FOLD_MIN_OUTPUT		:REAL	:=200.0;	//	翻板折弯比例阀最小起跳量_初始值
	CNST_HYD_CLAMP_ACC_STEP				:REAL	:=60.0;	//	夹钳比例阀加速步长_初始值
	CNST_HYD_CLAMP_DEC_STEP				:REAL	:=90.0;	//	夹钳比例阀减速步长_初始值
	CNST_HYD_CLAMP_MIN_OUTPUT			:REAL	:=180.0;	//	夹钳比例阀最小起跳量_初始值
							
	CNST_APRON_TOPSLIDE_FWD_SPD			:REAL	:=0.0;	//	上翻板滑动，前进，工作速度
	CNST_APRON_TOPSLIDE_FWD_CREEP_SPD	:REAL	:=0.0;	//	上翻板滑动，前进，爬行速度
	CNST_APRON_TOPSLIDE_BWD_SPD			:REAL	:=0.0;	//	上翻板滑动，后退，工作速度
	CNST_APRON_TOPSLIDE_BWD_CREEP_SPD	:REAL	:=0.0;	//	上翻板滑动，后退，爬行速度
								
	CNST_APRON_BTMSLIDE_FWD_SPD			:REAL	:=0.0;	//	下翻板滑动，前进，工作速度
	CNST_APRON_BTMSLIDE_FWD_CREEP_SPD	:REAL	:=0.0;	//	下翻板滑动，前进，爬行速度
	CNST_APRON_BTMSLIDE_BWD_SPD			:REAL	:=0.0;	//	下翻板滑动，后退，工作速度
	CNST_APRON_BTMSLIDE_BWD_CREEP_SPD	:REAL	:=0.0;	//	下翻板滑动，后退，爬行速度
							
	CNST_APRON_TOPSLIDE_FWD_DecDis		:REAL	:=0.0;	//	上翻板滑动，前进，减速距离
	CNST_APRON_TOPSLIDE_BWD_DecDis		:REAL	:=0.0;	//	上翻板滑动，后退，减速距离
	CNST_APRON_BTMSLIDE_FWD_DecDis		:REAL	:=0.0;	//	下翻板滑动，前进，减速距离
	CNST_APRON_BTMSLIDE_BWD_DecDis		:REAL	:=0.0;	//	下翻板滑动，后退，减速距离
	CNST_APRON_SLIDE_WINDOWS			:REAL	:=0.0;	//	翻板滑动，停止窗口
	CNST_APRON_TOPSLIDE_POS0			:REAL	:=0.0;	//	上翻板滑动，位置0
	CNST_APRON_TOPSLIDE_POS1			:REAL	:=0.0;	//	上翻板滑动，位置1
	CNST_APRON_TOPSLIDE_POS2			:REAL	:=0.0;	//	上翻板滑动，位置2
	CNST_APRON_TOPSLIDE_POS3			:REAL	:=0.0;	//	上翻板滑动，位置3
	CNST_APRON_BTMSLIDE_POS0			:REAL	:=0.0;	//	上翻板滑动，位置0
	CNST_APRON_BTMSLIDE_POS1			:REAL	:=0.0;	//	上翻板滑动，位置1
	CNST_APRON_BTMSLIDE_POS2			:REAL	:=0.0;	//	上翻板滑动，位置2
	CNST_APRON_BTMSLIDE_POS3			:REAL	:=0.0;	//	上翻板滑动，位置3
							
	CNST_APRON_TOPFOLD_FWD_SPD			:REAL	:=0.0;	//	上翻板折弯，前进，工作速度
	CNST_APRON_TOPFOLD_FWD_CREEP_SPD	:REAL	:=0.0;	//	上翻板折弯，前进，爬行速度
	CNST_APRON_TOPFOLD_BWD_SPD			:REAL	:=0.0;	//	上翻板折弯，后退，工作速度
	CNST_APRON_TOPFOLD_BWD_CREEP_SPD	:REAL	:=0.0;	//	上翻板折弯，后退，爬行速度
	CNST_APRON_BTMFOLD_FWD_SPD			:REAL	:=0.0;	//	下翻板折弯，前进，工作速度
	CNST_APRON_BTMFOLD_FWD_CREEP_SPD	:REAL	:=0.0;	//	下翻板折弯，前进，爬行速度
	CNST_APRON_BTMFOLD_BWD_SPD			:REAL	:=0.0;	//	下翻板折弯，后退，工作速度
	CNST_APRON_BTMFOLD_BWD_CREEP_SPD	:REAL	:=0.0;	//	下翻板折弯，后退，爬行速度
							
	CNST_APRON_TOPFOLD_FWD_DecDis_GT110	:REAL	:=0.0;	//	上翻板折弯，前进，>110度时，减速距离
	CNST_APRON_TOPFOLD_FWD_DecDis_LE110	:REAL	:=0.0;	//	上翻板折弯，后退，≤110度时，减速距离
	CNST_APRON_TOPFOLD_BWD_DecDis		:REAL	:=0.0;	//	上翻板折弯，后退，减速距离
	CNST_APRON_BTMFOLD_FWD_DecDis_GT110	:REAL	:=0.0;	//	下翻板折弯，前进，>110度时，减速距离
	CNST_APRON_BTMFOLD_FWD_DecDis_LE110	:REAL	:=0.0;	//	下翻板折弯，前进，≤110度时，减速距离
	CNST_APRON_BTMFOLD_BWD_DecDis		:REAL	:=0.0;	//	下翻板折弯，后退，减速距离
	CNST_APRON_FOLD_WINDOWS				:REAL	:=0.0;	//	翻板折弯，停止窗口
	CNST_APRON_TOPFOLD_MIN				:REAL	:=0.0;	//	上翻板折弯，最小极限
	CNST_APRON_TOPFOLD_MAX				:REAL	:=0.0;	//	上翻板折弯，最大极限
	CNST_APRON_BTMFOLD_MIN				:REAL	:=0.0;	//	下翻板折弯，最小极限
	CNST_APRON_BTMFOLD_MAX				:REAL	:=0.0;	//	下翻板折弯，最大极限
						
	CNST_CLAMP_OPEN_SPD_LT_HALF			:REAL	:=0.0;	//	钳口打开速度，低于半钳口位（手动模式）
	CNST_CLAMP_OPEN_SPD_GT_HALF			:REAL	:=0.0;	//	钳口打开速度，高于半钳口位
	CNST_CLAMP_CLOSE_SPD_LT_HALF		:REAL	:=0.0;	//	钳口下降速度，低于半钳口位
	CNST_CLAMP_CLOSE_SPD_GT_HALF		:REAL	:=0.0;	//	钳口下降速度，高于半钳口位
	CNST_CLAMP_LIGHT_PRESSURE_SETPOINT	:REAL	:=0.0;	//	钳口压紧时的压力值_轻型
	CNST_CLAMP_HEAVY_PRESSURE_SETPOINT	:REAL	:=0.0;	//	钳口压紧时的压力值_重型
	CNST_CLAMP_POS_CLOSED				:REAL	:=0.0;	//	钳口闭合位置
								
	CNST_BACKGAUGE_SPEED_HIGH			:REAL	:=0.0;	//	后夹送速度_高速
	CNST_BACKGAUGE_SPEED_LOW			:REAL	:=0.0;	//	后夹送速度_低速
	CNST_BACKGAUGE_ATTACH_PUSH			:REAL	:=0.0;	//	后夹送位置附加值_推动
	CNST_BACKGAUGE_ATTACH_GRIP			:REAL	:=0.0;	//	后夹送位置附加值_浅夹
	CNST_BACKGAUGE_ATTACH_OVERGRIP		:REAL	:=0.0;	//	后夹送位置附加值_深夹
	CNST_BACKGAUGE_ATTACH_BACK			:REAL	:=0.0;	//	后夹送位置附加值_后退
							
	CNST_TABLE_SPEED_HIGH				:REAL	:=0.0;	//	桌板速度_高速
	CNST_TABLE_POS_MAX					:REAL	:=0.0;	//	桌板限定位置_最大值
	CNST_TABLE_POS_MIN					:REAL	:=0.0;	//	桌板限定位置_最小值
								
	CNST_SLITTER_FWD_SPD				:REAL	:=0.0;	//	纵切前进，工作速度
	CNST_SLITTER_FWD_CREEP_SPD			:REAL	:=0.0;	//	纵切前进，爬行速度
	CNST_SLITTER_BWD_SPD				:REAL	:=0.0;	//	纵切后退，工作速度
	CNST_SLITTER_BWD_CREEP_SPD			:REAL	:=0.0;	//	纵切后退，爬行速度
								
	CNST_ANGLE_LIMIT_HEAVY				:REAL	:=0.0;	//	最大限制角度 重型
	CNST_ANGLE_LIMIT_LIGHT				:REAL	:=0.0;	//	最大限制角度 轻型
								
	CNST_LUBE_HYP_COUNTS				:REAL	:=0.0;	//	润滑泵注油动作计数
	CNST_LUBE_DURATION_WORK				:REAL	:=0.0;	//	润滑泵注油持续时间
	
	CNST_FEED_SPEED_HIGH				:INT	:=200;
	CNST_FEED_SPEED_LOW					:INT	:=50;
	CNST_FEED_SPEED_CREEP				:INT	:=20;
	CNST_FEED_POS_ZERO					:INT	:=0;
	CNST_FEED_POS_NegPlus				:INT	:=-20;
	CNST_FEED_POS_Window				:REAL	:=2.0;
	CNST_FEED_POS_MAX					:INT	:=5000;
	CNST_FEED_POS_MIN					:INT	:=-1000;
	
//	CNST_TAPER_REF_T1					:REAL	:=700.0;	//	锥度折弯 基准-T1距离
//	CNST_TAPER_REF_T2					:REAL	:=1460.0;	//	锥度折弯 基准-T2距离
//	CNST_TAPER_REF_T3					:REAL	:=2200.0;	//	锥度折弯 基准-T3距离
//	CNST_TAPER_REF_T4					:REAL	:=2960.0;	//	锥度折弯 基准-T4距离

	CNST_TAPER_REF						:REAL;
	CNST_TAPER_REF_T1					:REAL;
	CNST_TAPER_REF_T2					:REAL;
	CNST_TAPER_REF_T3					:REAL;
	CNST_TAPER_REF_T4					:REAL;

END_VAR

// ---- GVLs/GVL_IO.TcGVL

VAR_GLOBAL
(*------------------------------------------------Input Points-----------------------------------------*)
(*1st    EL1008  *)							
	In_pedal1_UnClamp		AT %I*		:BOOL;	(*脚踏1 -钳口放松*)
	In_pedal1_Clamp			AT %I*		:BOOL;	(*脚踏1 -钳口夹紧*)
	In_pedal1_Slitter		AT %I*		:BOOL;	(*脚踏1 -拉刀*)
	In_pedal1_SlitterBack	AT %I*		:BOOL;	(*脚踏1 -拉刀返回*)
	In_pedal1_Fold			AT %I*		:BOOL;	(*脚踏1 -折弯*)
	In_pedal1_Gripper		AT %I*		:BOOL;	(*脚踏1 -后定位夹钳*)
	In_swOperator			AT %I*		:BOOL;	(*操作员开/关*)
	In_btnReset				AT %I*		:BOOL;	(*复位*)
//(*2nd    EL1008  *)							
//	In_pedal_Autostart		AT %I*		:BOOL;	//开始折板	
//	In_bak11				AT %I*		:BOOL;	
//	In_bak12				AT %I*		:BOOL;	
//	In_bak13				AT %I*		:BOOL;	
//	In_bak14				AT %I*		:BOOL;	
//	In_bak15				AT %I*		:BOOL;	
//	In_bak16				AT %I*		:BOOL;	
//	In_bak17				AT %I*		:BOOL;	
(*3rd    EL1008  *)							
	In_sigSlitLmt0			AT %I*		:BOOL;	(*拉刀原点停止接近开关 *)
	In_sigSlitSlw0			AT %I*		:BOOL;	(*拉刀原点慢速接近开关*)
	In_sigSlitSlw1			AT %I*		:BOOL;	(*拉刀前进慢速接近开关*)
	In_sigSlitLmt1			AT %I*		:BOOL;	(*拉刀前进停止接近开关*)
	In_sigTopApron_FoldHome	AT %I*		:BOOL;	(*上翻板折弯原点接近开关*)
	In_sigTopApron_SlideFWD	AT %I*		:BOOL;	(*上翻板滑动前进接近开关*)
	In_sigBtmApron_FoldHome	AT %I*		:BOOL;	(*下翻板折弯原点接近开关*)
	In_sigBtmApron_SlideFWD	AT %I*		:BOOL;	(*下翻板滑动前进接近开关*)
(*4th    EL1008  *)							
	In_sigClampMute			AT %I*		:BOOL;	(*钳口静音接近开关 *)
	In_sigGaugingFrnt		AT %I*		:BOOL;	(*板厚接近开关1*)
	In_sigGaugingMid		AT %I*		:BOOL;	(*板厚接近开关2*)
	In_sigGaugingRear		AT %I*		:BOOL;	(*板厚接近开关3*)
	In_sigBoardPresent		AT %I*		:BOOL;	(*有板检测*)
	In_bak35				AT %I*		:BOOL;	(*备用2*)
	In_SigSheetDetect1		AT %I*		:BOOL;	(*板材检测1*)
	In_SigSheetDetect2		AT %I*		:BOOL;	(*板材检测2*)
//(*5th   EL1008  *)							
//	In_bak40				AT %I*		:BOOL;	
//	In_bak41				AT %I*		:BOOL;	
//	In_bak42				AT %I*		:BOOL;	
//	In_bak43				AT %I*		:BOOL;	
//	In_bak44				AT %I*		:BOOL;	
//	In_bak45				AT %I*		:BOOL;	
//	In_bak46				AT %I*		:BOOL;	
//	In_bak47				AT %I*		:BOOL;	
(*6th    EL1008  *)							
	In_swLC_Enable			AT %I*		:BOOL;	(*激光光幕校准开/关 *)
	In_sigLaserFinger		AT %I*		:BOOL;	(*激光传感器*)
	In_sigLC_VShort			AT %I*		:BOOL;	(*垂直光幕（短）*)
	In_sigLC_VLong			AT %I*		:BOOL;	(*垂直光幕（长）*)
	In_sigLC_H				AT %I*		:BOOL;	(*水平光幕*)
	In_EMG_RopeStop			AT %I*		:BOOL;	(*拉绳限位*)
	In_sigPumpJam			AT %I*		:BOOL;	(*油泵堵塞报警*)
	In_sigLubeJam			AT %I*		:BOOL;	(*润滑堵塞报警*)
(*7th    EL1008  *)							
	In_EMG_MainCabinet		AT %I*		:BOOL;	(*操作台急停*)
	In_EMG_HandleCabinet	AT %I*		:BOOL;	(*主控柜急停*)
	In_PowerON				AT %I*		:BOOL;	(*电源启动*)
	In_VltA_Running			AT %I*		:BOOL;	(*油泵变频A启动*)
	In_VltB_Running			AT %I*		:BOOL;	(*油泵变频B启动*)
	In_Vlt_Alarm			AT %I*		:BOOL;	(*变频无报警*)
	In_PumpLow_Alarm		AT %I*		:BOOL;	(*油泵液位低*)
	In_VltSlitter_Running	AT %I*		:BOOL;	(*拉刀变频启动*)

(*------------------------------------------------Output Points-----------------------------------------*)
(*1st    EL2008  *)
	Out_ApronBtm_SlideFWD	AT %Q*		:BOOL;	(*下翻板滑动前移*)
	Out_ApronBtm_SlideBWD	AT %Q*		:BOOL;	(*下翻板滑动后移*)
	Out_ApronBtm_FoldFWD	AT %Q*		:BOOL;	(*下翻板折弯前进*)
	Out_ApronBtm_FoldBWD	AT %Q*		:BOOL;	(*下翻板折弯返回*)
	Out_ApronTop_SlideFWD	AT %Q*		:BOOL;	(*上翻板滑动前移*)
	Out_ApronTop_SlideBWD	AT %Q*		:BOOL;	(*上翻板滑动后移*)
	Out_ApronTop_FoldFWD	AT %Q*		:BOOL;	(*上翻板折弯前进*)
	Out_ApronTop_FoldBWD	AT %Q*		:BOOL;	(*上翻板折弯返回*)
(*2nd    EL2008  *)							
	Out_ClampUp				AT %Q*		:BOOL;	(*钳口放松*)
	Out_ClampDown			AT %Q*		:BOOL;	(*钳口夹紧*)
	Out_SuctionCup1Vent		AT %Q*		:BOOL;	(*上料吸盘1放气*)
	Out_SuctionCup1Suction	AT %Q*		:BOOL;	(*上料吸盘1吸气*)
	Out_PumpB_Load_Ligh		AT %Q*		:BOOL;	(*泵B卸荷-轻型*)	
	Out_PumpB_Load_Heav		AT %Q*		:BOOL;	(*泵B卸荷-重型*)	
	Out_PumpA_Load_Ligh		AT %Q*		:BOOL;	(*泵A卸荷-轻型*)	
	Out_PumpA_Load_Heav		AT %Q*		:BOOL;	(*泵A卸荷-重型*)
(*3rd    EL2008  	Q2.x	*)
	Out_GaugingF_Ext		AT %Q*		:BOOL;	(*板厚调整油缸1伸出*)
	Out_GaugingF_Rtn		AT %Q*		:BOOL;	(*板厚调整油缸1缩回*)
	Out_GaugingR_Ext		AT %Q*		:BOOL;	(*板厚调整油缸2伸出*)
	Out_GaugingR_Rtn		AT %Q*		:BOOL;	(*板厚调整油缸2缩回*)
	Out_Gripper				AT %Q*		:BOOL;	(*后定位夹钳气缸夹紧*)
	Out_Gripper2			AT %Q*		:BOOL;	(*后定位夹钳气缸夹紧2*)
	Out_GripperDatum_S0		AT %Q*		:BOOL;	(*挡板气缸1伸出*)
	Out_GripperDatum_S1		AT %Q*		:BOOL;	(*挡板气缸2伸出*)
	(*
	Out_GripperDatum_S0  Out_GripperDatum_S1
       FALSE               FALSE           HOME
       TRUE                FALSE           PUSH
       FALSE               TRUE            GRIP
       TRUE                TRUE            OVERGRIP
	 *)
(*4th    EL2008  *)							
	Out_PumpA_ST			AT %Q*		:BOOL;	(*油泵A正转 *)
	Out_PumpB_ST			AT %Q*		:BOOL;	(*油泵B正转*)
	Out_SlitterFwd			AT %Q*		:BOOL;	(*拉刀正转*)
	Out_SlitterBwd			AT %Q*		:BOOL;	(*拉刀反转*)
	Out_SlitterSpeed		AT %Q*		:BOOL;	(*拉刀高低速*)
	Out_LubePump			AT %Q*		:BOOL;	(*润滑泵*)	
	Out_SuctionCup2Vent		AT %Q*		:BOOL;	(*上料吸盘2放气*)
	Out_SuctionCup2Suction	AT %Q*		:BOOL;	(*上料吸盘2吸气*)
(*5th    EL2008  *)							
	Out_OpLed_Red			AT %Q*		:BOOL;	(*操作员指示灯（红色）*)
	Out_OpLed_Yellow		AT %Q*		:BOOL;	(*操作员指示灯（黄色）*)	
	Out_OpLed_Green			AT %Q*		:BOOL;	(*操作员指示灯（绿色）*)
	Out_OpLed_Beep			AT %Q*		:BOOL;	(*操作员指示灯蜂鸣器*)
	Out_Led_Red				AT %Q*		:BOOL;	(*灯条(红色)*)	
	Out_Led_Yellow			AT %Q*		:BOOL;	(*灯条(黄色)*)
	Out_Led_Green			AT %Q*		:BOOL;	(*灯条(绿色)*)
	Out_Gripper3			AT %Q*		:BOOL;	(*后定位夹钳气缸夹紧3*)
(*6th    EL2008  *)							
	Out_FlipCupVent1		AT %Q*		:BOOL;	(*翻转吸盘放气*)
	Out_FlipCupSuction1		AT %Q*		:BOOL;	(*翻转吸盘吸气*)
	Out_FlipCupVent2		AT %Q*		:BOOL;	(*翻转吸盘放气*)
	Out_FlipCupSuction2		AT %Q*		:BOOL;	(*翻转吸盘吸气*)
	Out_bak54				AT %Q*		:BOOL;	(*备用*)
	Out_bak55				AT %Q*		:BOOL;	(*备用*)
	Out_bak56				AT %Q*		:BOOL;	(*备用*)
	Out_EMG_RopeStop		AT %Q*		:BOOL;	(*拉绳急停断电*)


	
(*------------------------------------------------ANALOG_in and out-----------------------------------------*)
	(*1th    EL3004  *)
	ANALOG_in_TopApronFold		AT %I*	:INT;	(*上翻板角度-位移传感器*)
	ANALOG_in_TopApronSlide		AT %I*	:INT;	(*上翻板滑动-位移传感器*)
	ANALOG_in_BtmApronFold		AT %I*	:INT;	(*下翻板角度-位移传感器*)
	ANALOG_in_BtmApronSlide		AT %I*	:INT;	(*下翻板滑动-位移传感器*)
	(*2th    EL3004  *)
	ANALOG_in_ClampHeight		AT %I*	:INT;	(*钳口高度    位移传感器*)
	ANALOG_in_PumpPress			AT %I*	:INT;	(*压力传感器*)
	ANALOG_in_bak23				AT %I*	:INT;	
	ANALOG_in_bak24				AT %I*	:INT;
	(*1th    EL4004  *)
	ANALOG_out_PumpA			AT %Q*	:INT;	(*油泵A调速*)
	ANALOG_out_PumpB			AT %Q*	:INT;	(*油泵B调速*)
	ANALOG_out_bak3				AT %Q*	:INT;
	ANALOG_out_bak4				AT %Q*	:INT;
	(*EL4024 4-20mA 比例阀输出*)
	ANALOG_out_BtmApronSlide	AT %Q*	:INT;	(*下翻板滑动比例阀 Term41 Ch2*)
	ANALOG_out_BtmApronFold		AT %Q*	:INT;	(*下翻板折弯比例阀 Term41 Ch1*)
	ANALOG_out_ClampUp			AT %Q*	:INT;	(*钳口放松比例阀 Term42 Ch2*)
	ANALOG_out_ClampDown		AT %Q*	:INT;	(*钳口夹紧比例阀 Term42 Ch1*)
	ANALOG_out_TopApronSlide	AT %Q*	:INT;	(*上翻板滑动比例阀 Term42 Ch4*)
	ANALOG_out_TopApronFold		AT %Q*	:INT;	(*上翻板折弯比例阀 Term42 Ch3*)
	(*1th    EL3024  *)
	ANALOG_in_PumpTemp			AT %I*	:INT;	(*油箱温度*)
	ANALOG_in_LiquidHeight		AT %I*	:INT;	(*液位高度*)
	ANALOG_in_bak43				AT %I*	:INT;	
	ANALOG_in_bak44				AT %I*	:INT;	
	
	(*Output AT %Q*: ARRAY [1..7, 1..8] OF BOOL;
	Input AT %I*: ARRAY [1..7, 1..8] OF BOOL;*)
END_VAR

// ---- POUs/MAIN.TcPOU
PROGRAM MAIN
VAR_EXTERNAL
	SysInfo													: SystemInfoCtrl;	 //Show online the global Sysinfo 
END_VAR
VAR
	TaskInfo												:	TaskInfoCtrl;
	bExecuteComplete			: BOOL;									//Command Execute Complete, not defined
	fbMachine:fbMachine;
	
	nStateCommandCheck: INT;
	
	fbVisu						: FB_Visu;		
	nCounter: INT;
	iBoot: INT;
	bBoot: BOOL;
	fbTon :TON;
	fbWritePersistentValue: WritePersistentData;
	i10 	:DINT;
	iModeSW: INT;
	ton1,ton2,ton3,ton4 :TON;
	B1: BOOL;
	i110: INT := 0;
	
	test1	:INPUT;
	test2: BOOL;
	rtTest2: R_trig;
	iAdd: INT;

END_VAR

TaskInfo();	
Boot();
ModeSw();

//Checking the Statecommands
CASE nStateCommandCheck OF
0:
	
	IF NOT FALSE THEN
		nStateCommandCheck:= 1;
	ELSE
		nStateCommandCheck:= 2;
	END_IF
	
1:
	IF PackTags.Command.CntrlCmd = ePMLCommand_Clear		
	  AND fbMachine.eState = ePMLState_Aborted	THEN
			fbMachine.eCommand	:= ePMLCommand_Clear;
	ELSIF PackTags.Command.CntrlCmd = ePMLCommand_Reset		
	  AND (fbMachine.eState = ePMLState_Stopped OR fbMachine.eState = ePMLState_Complete) THEN
			fbMachine.eCommand	:= ePMLCommand_Reset;
	ELSIF PackTags.Command.CntrlCmd = ePMLCommand_Start	
	  AND (fbMachine.eState = ePMLState_Idle OR (stPMLUnitModeConfiguration[fbMachine.eMode].aStateDisabled[ePMLState_Idle] AND fbMachine.eState = ePMLState_Stopped))
	  AND (NOT (PackTags.Command.Parameter[2].Value <= 0) OR NOT (fbMachine.eMode = 1))THEN
			fbMachine.eCommand	:= ePMLCommand_Start; 
	ELSIF PackTags.Command.CntrlCmd = ePMLCommand_Hold		
	  AND fbMachine.eState = ePMLState_Execute	
	  AND( fbMachine.eMode =  1 OR fbMachine.eMode =  4 OR fbMachine.eMode = 2)  THEN
			 fbMachine.eCommand	:= ePMLCommand_Hold;
	ELSIF PackTags.Command.CntrlCmd = ePMLCommand_Suspend	
	  AND fbMachine.eState = ePMLState_Execute	
	  AND (fbMachine.eMode = 4 OR fbMachine.eMode = 1)THEN
			 fbMachine.eCommand	:= ePMLCommand_Suspend;
	ELSIF PackTags.Command.CntrlCmd = ePMLCommand_Unhold	
	  AND fbMachine.eState = ePMLState_Held		THEN
			 fbMachine.eCommand	:= ePMLCommand_Unhold;
	ELSIF PackTags.Command.CntrlCmd = ePMLCommand_Unsuspend	
	  AND fbMachine.eState = ePMLState_Suspended	THEN
			 fbMachine.eCommand	:= ePMLCommand_Unsuspend;
	ELSIF PackTags.Command.CntrlCmd = ePMLCommand_Abort	THEN
			fbMachine.eCommand	:= ePMLCommand_Abort;
	ELSIF PackTags.Command.CntrlCmd = ePMLCommand_Stop	THEN
			fbMachine.eCommand	:= ePMLCommand_Stop;
	END_IF
	nStateCommandCheck:=0;
	
2:
	fbMachine.eCommand	:= ePMLCommand_Abort;
	IF fbMachine.eState = ePMLState_Aborted AND PackTags.Command.CntrlCmd = ePMLCommand_Clear THEN
		nStateCommandCheck:=1;
	END_IF
END_CASE

bButtonProductionReq := PackTags.Command.UnitMode = ePMLProtUnitMode_Production AND PackTags.Status.UnitModeCurrent <> PackTags.Command.UnitMode;

(*
fbMachine(
	eModeCommand:=PackTags.Command.UnitMode , 
	eCommand:=PackTags.Command.CntrlCmd , 
	eMode=>PackTags.Status.UnitModeCurrent , 
	eState=>PackTags.Status.StateCurrent , 
	bUndefinedDone=> , 
	bInvalidModeCommandOut=> , 
	bChangeIntoProduction=> );
	*)
fbMachine(eModeCommand:= PackTags.Command.UnitMode,  eMode => PackTags.Status.UnitModeCurrent, eState =>PackTags.Status.StateCurrent);
	
/// PackTags.Command.UnitModeChangeRequest;


  (* states according to PackTags v3.0 *)
  (*
    ePMLCommand_Undefined   := 0,
    ePMLCommand_Reset       := 1,
    ePMLCommand_Start       := 2,
    ePMLCommand_Stop        := 3,
    ePMLCommand_Hold        := 4,
    ePMLCommand_Unhold      := 5,
    ePMLCommand_Suspend     := 6,
    ePMLCommand_Unsuspend   := 7,
    ePMLCommand_Abort       := 8,
    ePMLCommand_Clear       := 9
	*)
	
M_Visu();

fbTon(IN:= NOT fbTon.Q , PT:=T#6S , Q=> , ET=> );
fbWritePersistentValue(
	NETID:='' ,
	PORT:= 851,
	START:=fbTon.Q ,
	TMOUT:=T#3s ,
	BUSY=> ,
	ERR=> ,
	ERRID=> );
IF fbTon.Q THEN
	i10:=i10+1;
END_IF;

(* Systemfunctions **********************************************************)
	SysInfo(
	RST:= , 
	RTCSyncCylce:=  , 
	TimeStampTrig:= pulse._100ms.RT , 
	ObjId=> , 
	TaskCnt=> , 
	OnlineChangeCount=> , 
	AppName=> , 
	AppTimestamp=> , 
	BootDataLoaded=> , 
	OldBootData=> , 
	TimeStampDT=> , 
	TimeStamp=> , 
	TimeStr=> , 
	DateStr=> , 
	TimeStamp2=> , 
	TimeStruct=> , 
	MonthDays=> , 
	LeapYear=> , 
	WeekOfYear=> , 
	timezoneId=> );

	Pulse();

	
	
	
	rtTest2(CLK:=Test2 , Q=> );
	test1(
	Force:= , 
	Invert:= , 
	PT_ON:=T#0S , 
	PT_OFF:=T#2S , 
	INPUT:=Test2 , 
	Q=> , 
	Q_RT=> , 
	Q_FT=> , 
	Q_DIRECT=> );

ACTION Boot:
(*
CASE iBoot OF
0:
iBoot	:=iBoot+1;
bBoot	:=TRUE;
1:	iBoot	:=iBoot+1;
2:	iBoot	:=iBoot+1;
3:	iBoot	:=iBoot+1;
4:	iBoot	:=iBoot+1;
5:
bBoot	:=FALSE;
RETURN;
END_CASE
*)
IF NOT TaskInfo.FirstCycle THEN
	RETURN;
END_IF

(*------------------------------------开机首次运行程序--------------------------*)
GVL.FirstDualPump_5m	:=TRUE;
Hmi_bArray[0]	:=stFolderPara.swSimplexDuplex;
Hmi_bArray[1]	:=stFolderPara.swLightHeavy;
Hmi_bArray[2]	:=stFolderPara.swSlitterVelocity;
Hmi_bArray[3]	:=stFolderPara.swLoadingTable;
Hmi_bArray[4]	:=stFolderPara.swAngleDisplay;
Hmi_bArray[5]	:=stFolderPara.swClampOpen_InManual;
Hmi_bArray[6]	:=stFolderPara.swClampOpen_InAuto;
Hmi_bArray[7]	:=stFolderPara.swFeedMechanism;

Hmi_rArray[50]	:=stFolderPara.SetFoldAngle;
Hmi_rArray[51]	:=stFolderPara.SetMoveBackgauge;
Hmi_rArray[52]	:=stFolderPara.SetTopApronSlide;
Hmi_rArray[53]	:=stFolderPara.SetBtmApronSlide;
Hmi_rArray[54]	:=stFolderPara.SetLoadingTable;



Hmi_rArray[100]	:=stFolderPara.Clamp_LowPos;
Hmi_rArray[101]	:=stFolderPara.Clamp_MidPos;
Hmi_rArray[102]	:=stFolderPara.Clamp_HighPos;
Hmi_rArray[103]	:=stFolderPara.Clamp_MaxPos;
Hmi_rArray[104]	:=stFolderPara.ClampHalfPos;
Hmi_rArray[105]	:=stFolderPara.Clamp_PressFlat;
Hmi_rArray[106]	:=stFolderPara.Clamp_FoldEnd;

Hmi_rArray[110]	:=stFolderPara.BackgaugeMaxPos;
Hmi_rArray[111]	:=stFolderPara.BackgaugeMinPos;
Hmi_rArray[112]	:=stFolderPara.SlitterOffset;
Hmi_rArray[113]	:=stFolderPara.BtmApronZeroPosition;
Hmi_rArray[114]	:=stFolderPara.TopApronZeroPosition;
Hmi_rArray[115]	:=stFolderPara.SquashBackstop_Top;
Hmi_rArray[116]	:=stFolderPara.SquashBackstop_Btm;
Hmi_rArray[117]	:=stFolderPara.SquashBackstop_External;
Hmi_rArray[118]	:=stFolderPara.SquashBackstop_OpenTop;
Hmi_rArray[119]	:=stFolderPara.SquashBackstop_OpenBtm;

Hmi_rArray[120]	:=stFolderPara.MT1_BackstopZero;
Hmi_rArray[121]	:=stFolderPara.MT2_BackstopZero;
Hmi_rArray[122]	:=stFolderPara.MT3_BackstopZero;
Hmi_rArray[123]	:=stFolderPara.MT4_BackstopZero;



Hmi_rArray[94]	:=stFolderPara.Clamp_FeedPos;
Hmi_rArray[107]	:=stFolderPara.FeedOffset;
Hmi_rArray[108]	:=stFolderPara.FeedPosition;
Hmi_rArray[109]	:=stFolderPara.SetMoveFeed;

FOR iAdd:=0 TO 14 BY 1 DO
    Hmi_rArray[150+iAdd]:=stFolderPara.BtmAngleAddit[iAdd];
	Hmi_rArray[170+iAdd]:=stFolderPara.TopAngleAddit[iAdd];
END_FOR;


IF NOT stFolder.Taper_SW THEN
	stFolderCom.SpeedRatio_T1:=stFolderCom.SpeedRatio_T2:=
	stFolderCom.SpeedRatio_T3:=stFolderCom.SpeedRatio_T4:=1;
END_IF
END_ACTION

METHOD M_Visu : BOOL
VAR_INPUT
END_VAR
fbVisu(
	
	aKeyPressed:=aKeyPressed , 
	aUnitInfo:=aUnitInfo , 
	
	aCaption=> aCaption, 
	eModeVisu=> , 
	eStateVisu=> , 
	sUnitName=> , 
	iFrameVisible=> );
END_METHOD

ACTION ModeSw:
CASE iModeSW OF
0:
	IF NOT(PackTags.Command.UnitMode= UINT_TO_DINT(Hmi_iArray[0])) THEN
		IF PackTags.Status.UnitModeCurrent=0 THEN
			PackTags.Command.UnitModeChangeRequest	:=TRUE;
			PackTags.Command.UnitMode	:=Hmi_iArray[0];
			iModeSW	:=10;
		ELSE
			iModeSW	:=11;
		END_IF
	END_IF
10:
	IF PackTags.Status.StateCurrent=ePMLState_Aborted THEN
		PackTags.Command.CntrlCmd	:=ePMLCommand_Clear;
	ELSIF PackTags.Status.StateCurrent=ePMLState_Stopped THEN
		iModeSW:=11;
	END_IF;
11:
	PackTags.Command.CntrlCmd	:=ePMLCommand_Stop;
	IF PackTags.Status.StateCurrent=ePMLState_Stopped THEN
		PackTags.Command.UnitModeChangeRequest	:=TRUE;
		PackTags.Command.UnitMode	:=Hmi_iArray[0];
		iModeSW:=20;
	END_IF
20:
	IF PackTags.Status.UnitModeCurrent=Hmi_iArray[0] THEN
		PackTags.Command.UnitModeChangeRequest	:=FALSE;
		iModeSW:=21;
	END_IF
21:	
	PackTags.Command.CntrlCmd	:=ePMLCommand_Reset;
	IF PackTags.Status.StateCurrent=ePMLState_Idle THEN
		PackTags.Command.CntrlCmd	:=ePMLCommand_Start;
		iModeSW:=22;
	END_IF;
22:
	IF PackTags.Status.StateCurrent=ePMLState_Execute THEN
		iModeSW:=0;
	END_IF;
END_CASE
END_ACTION

END_PROGRAM

// ---- POUs/SystemInfo/SystemInfoCtrl.TcPOU
{attribute 'no_check'}
FUNCTION_BLOCK SystemInfoCtrl
VAR CONSTANT
	ENG_DATE_FORMAT											:	BOOL := TRUE;
END_VAR                     								
VAR_INPUT                   								
	RST														:	BOOL;
	RTCSyncCylce											:	DWORD := 5; (* in seconds *)
	TimeStampTrig											:	BOOL;
END_VAR
VAR_OUTPUT
//PlcAppSystemInfo
	ObjId													: 	OTCID;
	TaskCnt													: 	UDINT; //The number of tasks in the actual runtime system
	OnlineChangeCount										: 	UDINT;
	AppName													: 	STRING(63);
	AppTimestamp											:	DT;
	BootDataLoaded											: 	BOOL;
	OldBootData												: 	BOOL;
	
//General	
	TimeStampDT												:	DATE_AND_TIME;
	TimeStamp												:	STRING(25); (* DD.MM.YY-Stunde:Minute:Sekunde:xxx *)
	TimeStr													:	STRING(15);	(* hh.mm.ss.xxms *)
	DateStr													:	STRING(15);	(* mm.dd.jj *)
	TimeStamp2												:	STRING(25); (* YYYY-MM-DD_HHMMSS for example YYYY-MM-DD_HHMMSS_Name.txt *)
	TimeStruct												:	TIMESTRUCT;
	MonthDays												:	WORD;
	LeapYear												:	BOOL;
	WeekOfYear												:	WORD;
	timezoneId												: 	E_TimeZoneID;
END_VAR

VAR
	(* Inst. Get Taskindex *)
	InstGETCURTASKINDEX										: 	GETCURTASKINDEX;
	InstLocalSystemTime										:	FB_LocalSystemTime;
	_sec													:	WORD;
	_hour													:	WORD;
END_VAR

	(********************************************************************************)
	(*	(c) by Beckhoff Automation													*)
	(*																				*)
	(*		B E C K H O F F   N E W   A U T O M A T I O N   T E C H N O L O G Y     *)
	(*																				*)
	(*		Eiserstr.5	D-33415 Verl	Germany	phone:	+49-5246-0	www.Beckhoff.Com*)
    (*																				*)
    (*		Bausteinbeschreibung	: 	evaluate the PlcAppSystemInfo				*)
	(*									and get timestamp							*)
	(*																				*)
	(*		Version					:	V3.0										*)
	(*		Stand					:	03.2013										*)
 	(*		Autor					:	Daniel Schlingmann							*)
	(*																				*)
	(********************************************************************************)

(* Get Current Task Index ************************************************************************)
	IF InstGETCURTASKINDEX.index = 0 
	THEN 
		InstGETCURTASKINDEX(); 
	END_IF

(* Read System Info Current Task *****************************************************************)
	ObjId													:= TwinCAT_SystemInfoVarList._AppInfo.ObjId;
	TaskCnt 												:= TwinCAT_SystemInfoVarList._AppInfo.TaskCnt;
	OnlineChangeCount										:= TwinCAT_SystemInfoVarList._AppInfo.OnlineChangeCnt;
	AppName													:= TwinCAT_SystemInfoVarList._AppInfo.AppName;	
	AppTimestamp											:= TwinCAT_SystemInfoVarList._AppInfo.AppTimestamp;

	(* Retein/Persisten Data Err *)
	IF TwinCAT_SystemInfoVarList._TaskInfo[InstGETCURTASKINDEX.Index].FirstCycle 
	THEN
		BootDataLoaded										:= TwinCAT_SystemInfoVarList._AppInfo.BootDataLoaded;
		OldBootData											:= TwinCAT_SystemInfoVarList._AppInfo.OldBootData;
	ELSIF RST 
	THEN
		Reset();
	ELSE
		;
	END_IF

(* evalutate systemtime ************************************************************************)
	InstLocalSystemTime(
		sNetID		:= '',
		bEnable		:= TRUE,
		dwCycle		:= RTCSyncCylce,
		dwOpt		:= (* Default *),
		tTimeout	:= (* Default *),
		bValid		=> ,
		systemTime	=> TimeStruct,
		tzID		=> timezoneId);

	IF TimeStampTrig
		AND InstLocalSystemTime.bValid
	THEN
		(* Date dd.mm.jj ********************)
		IF TimeStruct.wDay < 10 
		THEN
			DateStr 										:= CONCAT('0',WORD_TO_STRING(TimeStruct.wDay));
		ELSE        										
			DateStr 										:= WORD_TO_STRING(TimeStruct.wDay);
		END_IF
		DateStr 											:= CONCAT(DateStr,'.');
		IF TimeStruct.wMonth < 10 
		THEN
			DateStr 										:= CONCAT(DateStr,CONCAT('0',WORD_TO_STRING(TimeStruct.wMonth)));
		ELSE        										
			DateStr 										:= CONCAT(DateStr,WORD_TO_STRING(TimeStruct.wMonth));
		END_IF
		
		DateStr 											:= CONCAT(DateStr,'.');
		DateStr 											:= CONCAT(DateStr,RIGHT(WORD_TO_STRING(TimeStruct.wYear),2));
	
		(* Time hh.mm.ss.xxms ***************)
		IF TimeStruct.wHour < 10 
		THEN
			TimeStr 										:= CONCAT('0',WORD_TO_STRING(TimeStruct.wHour));
		ELSE        										
			TimeStr 										:= WORD_TO_STRING(TimeStruct.wHour);
		END_IF
		
		TimeStr 											:= CONCAT(TimeStr,':');
		
		IF TimeStruct.wMinute < 10 
		THEN
			TimeStr 										:= CONCAT(TimeStr,CONCAT('0',WORD_TO_STRING(TimeStruct.wMinute)));
		ELSE
			TimeStr 										:= CONCAT(TimeStr,WORD_TO_STRING(TimeStruct.wMinute));
		END_IF
		
		TimeStr 											:= CONCAT(TimeStr,':');
		
		IF TimeStruct.wSecond < 10 
		THEN
			TimeStr 										:= CONCAT(TimeStr,CONCAT('0',WORD_TO_STRING(TimeStruct.wSecond)));
		ELSE        										
			TimeStr 										:= CONCAT(TimeStr,WORD_TO_STRING(TimeStruct.wSecond));
		END_IF      										
		
		TimeStr 											:= CONCAT(TimeStr,'.');
		TimeStr 											:= CONCAT(TimeStr,WORD_TO_STRING(TimeStruct.wMilliseconds));
		
		(* TimeStamp Format DE: DD.MM.YY-Stunde:Minute:Sekunde:xxx,*)
		TimeStamp 											:= CONCAT(DateStr,'-');
		TimeStamp 											:= CONCAT(TimeStamp,TimeStr);
		TimeStamp 											:= CONCAT(TimeStamp,':');
		
		IF TimeStruct.wMilliseconds > 100 
		THEN
			TimeStamp										:=CONCAT(TimeStamp,WORD_TO_STRING(TimeStruct.wMilliseconds));
		ELSIF TimeStruct.wMilliseconds > 10 
		THEN
			TimeStamp										:=CONCAT(CONCAT(TimeStamp,'0'),WORD_TO_STRING(TimeStruct.wMilliseconds));
		ELSE
			TimeStamp										:=CONCAT(CONCAT(TimeStamp,'00'),WORD_TO_STRING(TimeStruct.wMilliseconds));
		END_IF
	
		(* Timestamp Format ENG: YYYY-MM-DD-hh:mm:ss.xxx *)
		(* TimeStamp := SYSTEMTIME_TO_STRING(TimeStruct); *)
	
		(* TimeStamp2 FileName YYYY-MM-DD_HHMMSS *)
		IF _sec <> TimeStruct.wSecond 
		THEN
			
			TimeStamp2 										:= CONCAT(WORD_TO_STRING(TimeStruct.wYear),'-');
			
			IF TimeStruct.wMonth < 10 
			THEN
				TimeStamp2 									:= CONCAT(TimeStamp2,CONCAT('0',WORD_TO_STRING(TimeStruct.wMonth)));
			ELSE           									
				TimeStamp2 									:= CONCAT(TimeStamp2,WORD_TO_STRING(TimeStruct.wMonth));
			END_IF
			
			TimeStamp2 										:= CONCAT(TimeStamp2,'-');
			
			IF TimeStruct.wDay < 10 
			THEN
				TimeStamp2 									:= CONCAT(TimeStamp2,CONCAT('0',WORD_TO_STRING(TimeStruct.wDay)));
			ELSE           									
				TimeStamp2 									:= CONCAT(TimeStamp2,WORD_TO_STRING(TimeStruct.wDay));
			END_IF
			
			TimeStamp2 										:= CONCAT(TimeStamp2,'_');
			
			IF TimeStruct.wHour < 10 
			THEN
				TimeStamp2 									:= CONCAT(TimeStamp2,CONCAT('0',WORD_TO_STRING(TimeStruct.wHour)));
			ELSE           									
				TimeStamp2 									:= CONCAT(TimeStamp2,WORD_TO_STRING(TimeStruct.wHour));
			END_IF
			IF TimeStruct.wMinute < 10 
			THEN
				TimeStamp2 									:= CONCAT(TimeStamp2,CONCAT('0',WORD_TO_STRING(TimeStruct.wMinute)));
			ELSE           									
				TimeStamp2 									:= CONCAT(TimeStamp2,WORD_TO_STRING(TimeStruct.wMinute));
			END_IF
			IF TimeStruct.wSecond < 10 
			THEN
				TimeStamp2 									:= CONCAT(TimeStamp2,CONCAT('0',WORD_TO_STRING(TimeStruct.wSecond)));
			ELSE           									
				TimeStamp2 									:= CONCAT(TimeStamp2,WORD_TO_STRING(TimeStruct.wSecond));
			END_IF
			
			_sec 											:= TimeStruct.wSecond;
	
			(* information of year *)
			TimeStampDT 									:= SYSTEMTIME_TO_DT(TimeStruct);
			MonthDays										:= F_GetMaxMonthDays(TimeStruct.wYear,TimeStruct.wMonth);
			LeapYear										:= F_YearIsLeapYear(TimeStruct.wYear) ;
			WeekOfYear										:= F_GetWeekOfTheYear(TimeStampDT);
	
		END_IF
	END_IF

(**************************************************************************************************)

METHOD PUBLIC Reset
VAR_INPUT
END_VAR
OldBootData 												:= FALSE;
END_METHOD

END_FUNCTION_BLOCK

// ---- POUs/SystemInfo/TaskInfoCtrl.TcPOU
{attribute 'no_check'}
FUNCTION_BLOCK TaskInfoCtrl
VAR_INPUT
END_VAR
VAR_OUTPUT
	Index													:	INT := 1;
	TaskName          										: 	STRING(63);
	ObjId             										: 	OTCID;
	CycleTime         										: 	UDINT;
	CycleTimeMS       										: 	TIME;	
	CycleTimeFloat											:	LREAL;	
	Priority          										: 	UINT;
	AdsPort           										: 	UINT;
	CycleCount        										: 	UDINT;
	DcTaskTime        										: 	LINT;
	LastExecTime      										: 	UDINT;
	FirstCycle        										: 	BOOL;
	CycleTimeExceeded 										: 	BOOL;	
	CycleTimeExceededCount 									: 	UDINT;
END_VAR

VAR
	GETCURTASKINDEX		: GETCURTASKINDEX;
END_VAR

	(********************************************************************************)
	(*	(c) by Beckhoff Automation													*)
	(*																				*)
	(*		B E C K H O F F   N E W   A U T O M A T I O N   T E C H N O L O G Y     *)
	(*																				*)
	(*		Eiserstr.5	D-33415 Verl	Germany	phone:	+49-5246-0	www.Beckhoff.Com*)
    (*																				*)
    (*		Bausteinbeschreibung	: evaluate PlcTaskSystemInfo Arrays				*)
	(*																				*)
	(*		Version					:	V2.0										*)
	(*		Stand					:	03.2013										*)
 	(*		Autor					:	Daniel Schlingmann							*)
	(*																				*)
	(********************************************************************************)

(* Get Current Task Index ************************************************************************)
	IF GETCURTASKINDEX.index = 0 	
	THEN 
		GETCURTASKINDEX(index => index); 
		//Init
		TaskName          									:= TwinCAT_SystemInfoVarList._TaskInfo[index].TaskName;
		ObjId             									:= TwinCAT_SystemInfoVarList._TaskInfo[index].ObjId;
		CycleTime         									:= TwinCAT_SystemInfoVarList._TaskInfo[index].CycleTime;
		Priority          									:= TwinCAT_SystemInfoVarList._TaskInfo[index].Priority;
		AdsPort           									:= TwinCAT_SystemInfoVarList._TaskInfo[index].AdsPort;
		CycleTimeMS											:= LREAL_TO_TIME(UDINT_TO_LREAL(CycleTime) * 0.0001 );
		CycleTimeFloat										:= (UDINT_TO_LREAL(CycleTime) * 0.0001 / 1000.0);		
	END_IF

	//Cylic 
	CycleCount        										:= TwinCAT_SystemInfoVarList._TaskInfo[index].CycleCount;
	DcTaskTime        										:= TwinCAT_SystemInfoVarList._TaskInfo[index].DcTaskTime; 
	LastExecTime      										:= TwinCAT_SystemInfoVarList._TaskInfo[index].LastExecTime;
	FirstCycle        										:= TwinCAT_SystemInfoVarList._TaskInfo[index].FirstCycle;
	CycleTimeExceeded 										:= TwinCAT_SystemInfoVarList._TaskInfo[index].CycleTimeExceeded;
	IF CycleTimeExceeded 
	THEN
		CycleTimeExceededCount								:= CycleTimeExceededCount + 1;	
	END_IF

(**************************************************************************************************)

END_FUNCTION_BLOCK

// ---- POUs/PulseGenerator/PulseCtrl.TcPOU
FUNCTION_BLOCK PulseCtrl
VAR_INPUT
END_VAR
VAR_OUTPUT
	BlinkSlow												: 	BOOL;
	Blink													: 	BOOL;
	BlinkFast												: 	BOOL;
	BlinkVeryFast											:	BOOL;
	BlinkFlash												:	BOOL;
	
//	_20ms													: PulseGeneratorCtrl := (PT_OFF := T#20MS, 		PT_ON := T#20MS);
	_100ms													: PulseGeneratorCtrl := (PT_OFF := T#100MS, 		PT_ON := T#100MS);
	_250ms													: PulseGeneratorCtrl := (PT_OFF := T#250MS, 		PT_ON := T#250MS); (* Blink very Fast *)
	_400ms													: PulseGeneratorCtrl := (PT_OFF := T#400MS, 		PT_ON := T#400MS); (* Blink Fast *)
	_500ms													: PulseGeneratorCtrl := (PT_OFF := T#500MS, 		PT_ON := T#500MS);
	_800ms													: PulseGeneratorCtrl := (PT_OFF := T#800MS, 		PT_ON := T#800MS); (* Blink *)
	_1s														: PulseGeneratorCtrl := (PT_OFF := T#1S, 			PT_ON := T#1S);
	_1s600ms												: PulseGeneratorCtrl := (PT_OFF := T#1S600MS, 	PT_ON := T#1S600MS); (* Blink Slow *)
	_2s														: PulseGeneratorCtrl := (PT_OFF := T#2S, 			PT_ON := T#2S); 
	_5s														: PulseGeneratorCtrl := (PT_OFF := T#5S, 			PT_ON := T#5S);
//	_10s													: PulseGeneratorCtrl := (PT_OFF := T#10S, 		PT_ON := T#10S); 
//	_2m														: PulseGeneratorCtrl := (PT_OFF := T#2M, 			PT_ON := T#2M); 
	_5m														: PulseGeneratorCtrl := (PT_OFF := T#5M, 			PT_ON := T#5M); 
//	_30m													: PulseGeneratorCtrl := (PT_OFF := T#30m, 		PT_ON := T#30m); 
END_VAR
VAR
	_Flash													: PulseGeneratorCtrl := (PT_OFF := T#800MS, PT_ON := T#80MS); (* Blink Flash *)
END_VAR

(************************************************************************************************************)
(* function-block generates different 																		*)
(************************************************************************************************************)

(* impuls generator *****************************************************************************************)
	(* Blitz Takt *)
	_Flash(
		PT_OFF	:= ,
		PT_ON	:= ,
		Q		=> BlinkFlash,
		RT		=> );

	(* Generiere 20ms Takt *)
(*	_20ms(
		PT_OFF	:= ,
		PT_ON	:= ,
		Q		=> ,
		RT		=> ); *)

	(* Generiere 100ms Q *)
	_100ms(
		PT_OFF	:= ,
		PT_ON	:= ,
		Q		=> ,
		RT		=> );

	(* Generiere 250ms Q Flimmerlicht*)
	_250ms(
		PT_OFF	:= ,
		PT_ON	:= ,
		Q		=> BlinkVeryFast,
		RT		=> );

	(* Generiere 400ms Q Schnelles Blinklicht *)
	_400ms(
		PT_OFF	:= ,
		PT_ON	:= ,
		Q		=> BlinkFast,
		RT		=> ); 

	(* Generiere 500ms Q *)
	_500ms(
		PT_OFF	:= ,
		PT_ON	:= ,
		Q		=> ,
		RT		=> );

	(* Generiere 800ms Q Blinklicht *)
	_800ms(
		PT_OFF	:= ,
		PT_ON	:= ,
		Q		=> Blink, 
		RT		=> );

	(* Generiere 1s Q *)
	_1s(
		PT_OFF	:= T#1S,
		PT_ON	:= T#1S,
		Q		=> ,
		RT		=> );

	(* Generiere 1s600ms Q Langsames Blinklicht *)
	_1s600ms(
		PT_OFF	:= ,
		PT_ON	:= ,
		Q		=> BlinkSlow,
		RT		=> );

	(* Generiere 2s Q *)
	_2s(
		PT_OFF	:= T#2S,
		PT_ON	:= T#2S,
		Q		=> ,
		RT		=> ); 

	(* Generiere 2s Q *)
	_5s(
		PT_OFF	:= ,
		PT_ON	:= ,
		Q		=> ,
		RT		=> );

	(* Generiere 10s Q *)
(*	_10s(
		PT_OFF	:= ,
		PT_ON	:= ,
		Q		=> ,
		RT		=> ); *)

	(* Generiere 2Min Q *)
(*	_2m(
		PT_OFF	:= t#2m,
		PT_ON	:= t#2m,
		Q		=> ,
		RT		=> ); *)

	(* Generiere 5Min Q *)
	_5m(
		PT_OFF	:= T#5M,
		PT_ON	:= T#5M,
		Q		=> ,
		RT		=> ); 

	(* Generiere 30Min Q *)
(*	_30m(
		PT_OFF	:= ,
		PT_ON	:= ,
		Q		=> ,
		RT		=> ); *)

(************************************************************************************************)

END_FUNCTION_BLOCK

// ---- POUs/PulseGenerator/PulseGeneratorCtrl.TcPOU
FUNCTION_BLOCK PulseGeneratorCtrl
VAR_INPUT
	PT_OFF													: TIME;
	PT_ON													: TIME;
END_VAR             										
VAR_OUTPUT          										
	Q														: BOOL := FALSE;
	RT														: BOOL := FALSE;
END_VAR             										
VAR                 	
	TON_PULSE												: TON;
END_VAR

	(********************************************************************************)
	(*	(c) by Beckhoff Automation													*)
	(*																				*)
	(*		B E C K H O F F   N E W   A U T O M A T I O N   T E C H N O L O G Y    	*)
	(*																				*)
	(*		Eiserstr.5	D-33415 Verl	Germany	phone:	+49-5246-0	www.Beckhoff.Com*)
    (*																				*)
    (*		Bausteinbeschreibung	:	Taktgeber									*)
	(*		Version					:	V1.2										*)
	(*		Stand					:	01.2006										*)
 	(*		Autor					:	Daniel Schlingmann							*)
	(*																				*)
	(*********************************************************************************)

(* Reset Flanke *)
RT 															:= FALSE;
(* Taktgenerator *)
IF 	TON_PULSE.Q 
	AND Q 
THEN
	TON_PULSE(IN:=FALSE  , PT:= PT_OFF);
	RT 														:= Q;
	Q 														:= FALSE;
ELSIF	TON_PULSE.Q 
	AND NOT Q 
THEN
	RT 														:= NOT Q;
	TON_PULSE(IN:= FALSE , PT:= PT_ON) ;
	Q 														:= TRUE;
END_IF
(* Work Timer *)

TON_PULSE(IN:=TRUE);

(***********************************************************************************************************************)

END_FUNCTION_BLOCK

// ---- POUs/Actuators/Cylinder/CYLINDER.TcPOU
{attribute 'no_check'}
FUNCTION_BLOCK CYLINDER
VAR_INPUT  (* Peripherie Outputs *)
	InAck													:	BOOL;
	ToWorkPos												:	BOOL;
	ToBasePos												:	BOOL;
{attribute 'displaymode':='binary'}         			
	Options													:	BYTE  := 2#00000000;  (*
																		DISABLE_FEEDBACK_BP	= .0
																		DISABLE_FEEDBACK_WP	= .1
																		IMPULS_VALVE		= .7
																				*)
	FeedBasePos												:	BOOL := TRUE;
	FeedWorkPos												:	BOOL := TRUE;
	PT_Timeout												:	TIME := T#5S; (* Runtime check BasePos *)
	PT_Feedback												:	TIME := T#3S; (* Delay simulate Feedback *)
	RevStatusDirection										:	BOOL := FALSE;
END_VAR                                     			
VAR_OUTPUT  (* Peripherie Inputs *)         			
	I_BasePos												:	BOOL;
	I_Workpos												:	BOOL;
	Done													:	BOOL; (*	Endlage angefahren - nur aktiv wenn EIN Ausgang angesteuert und die Endlage erreicht ist *)
	Busy													:	BOOL;
	ErrBasePos												:	BOOL;
	ErrWorkPos												:	BOOL;
	ErrLogic												:	BOOL; (* Both Feedbacks signaled *)
{attribute 'displaymode':='binary'}         			
	Status													:	BYTE;	(* 	Bit 0 = Q_Grdst
																			Bit 1 = Q_Arbst
																			Bit 2 = I_Grdst
																			Bit 3 = I_Arbst
																			Bit 4 = Feed Grdst
																			Bit 5 = Feed Arbst
																			Bit 6 = BTB
																			Bit 7 = Error
																		*)
	Q_BasePos									(*	AT  %Q**) :	BOOL;
	Q_WorkPos									(*	AT  %Q* *):	BOOL;
END_VAR
VAR// IOs 
	SIG_BASEPOS												: INPUT;
	SIG_WORKPOS												: INPUT;
	TON_ErrWorkPos											: TON;
	TON_ErrBasePos											: TON;
END_VAR

	(* CylinderExt IO V2.4					 								             	 		*)
	(* Include functionblock "INPUT" 																*)
	(*********************************************************************************)

(* Write Output *****************************************************)
	IF ToBasePos AND ToWorkPos 
	THEN
		ON();
	ELSIF ToBasePos 	
	THEN
		BasePos();
	ELSIF ToWorkPos 
	THEN
		WorkPos();
	ELSE
		OFF();
	END_IF

(* Reedkontakte lesen ***********************************************)
	SIG_BASEPOS(
		Force	:= Q_BasePos AND NOT I_WorkPos AND Options.0,
		Invert	:= ,
		PT_ON	:= SEL(Options.0 ,T#0MS,PT_FEEDBACK),
		PT_OFF	:= ,
		Q_DIRECT=>,
		Q		=> I_BasePos,
		Q_RT	=> ,
		Q_FT	=> ,
		INPUT	=> );

	SIG_WORKPOS(
		Force	:= Q_WorkPos AND NOT I_BasePos AND Options.1,
		Invert	:= ,
		PT_ON	:= SEL(Options.1 ,T#0MS,PT_FEEDBACK),
		PT_OFF	:= ,
		Q_DIRECT=>,
		Q		=> I_WorkPos,
		Q_RT	=> ,
		Q_FT	=> ,
		INPUT	=> );
		
(* Status *************************************************)
	(* Move *)
	IF Q_BasePos AND NOT Q_WorkPos AND (NOT I_BasePos OR I_WorkPos)
	THEN
		Status.0 											:= NOT RevStatusDirection;
		Status.1											:= RevStatusDirection;
	ELSIF Q_WorkPos AND NOT Q_BasePos AND (NOT I_WorkPos OR I_BasePos)
	THEN
		Status.0											:= RevStatusDirection;
		Status.1											:= NOT RevStatusDirection;
	END_IF              									

	(* BasePos / WorkPos reached*)
	Status.2 												:= SEL(RevStatusDirection, I_BasePos , I_WorkPos);
	Status.3 												:= SEL(RevStatusDirection, I_WorkPos , I_BasePos);
 				        									
	(* not enabled*)    									
	Status.4 												:= SEL(RevStatusDirection, FeedBasePos , FeedWorkPos);
	Status.5 												:= SEL(RevStatusDirection, FeedWorkPos , FeedBasePos);
                        									
	(* Ready *)         									
	Status.6												:= NOT Status.7; 
	                    									
	(* Error *)         									
	Status.7 												:= ErrBasePos OR ErrWorkPos OR ErrLogic;
                        	
(* ack Error **********************************************************)
	IF InAck 
	THEN 
		ack(); 
	END_IF

(* Ueberwachung WorkPos ************************************************)
	TON_ErrWorkPos(	IN := Q_WorkPos
							AND (NOT I_WorkPos OR I_BasePos),
					PT := MAX(PT_Timeout,PT_Feedback + T#1S),
					Q => ErrWorkPos);

(* Ueberwachung WorkPos ************************************************)
	TON_ErrBasePos(	IN := Q_BasePos
							AND (NOT I_BasePos OR I_WorkPos),
					PT := MAX(PT_Timeout,PT_Feedback + T#1S),
					Q => ErrBasePos);

(*********************************************************************)

METHOD PUBLIC Ack
IF TON_ErrWorkPos.Q
	OR TON_ErrBasePos.Q
THEN
	TON_ErrWorkPos(IN := FALSE);
	TON_ErrBasePos(IN := FALSE);
ELSE
	; (* No error aktiv *)
END_IF

Status.7 													:= FALSE;
END_METHOD

METHOD PUBLIC BasePos : BOOL //Return = Done
ToWorkPos 													:= Q_WorkPos	:= FALSE;
ToBasePos 													:= TRUE;
Q_BasePos	 												:= FeedBasePos AND (NOT Options.7 OR NOT I_BasePos);
BasePos 													:= Done			:= I_BasePos;
Busy														:= NOT Done;
END_METHOD

METHOD PUBLIC Enable : BOOL //Return  Done - FALSE = BasePos , True = WorkPos
VAR_INPUT
	IN														:	BOOL;
END_VAR
IF IN
THEN
	Enable 													:= WorkPos();
ELSE
	Enable 													:= NOT BasePos();
END_IF
END_METHOD

METHOD PUBLIC OFF
Done 														:= Busy := Q_WorkPos := Q_BasePos := FALSE;
ToBasePos 													:= TOWorkPos := FALSE;
END_METHOD

METHOD PUBLIC ON
ToWorkPos 													:= Q_WorkPos 	:= FeedWorkPos;
ToBasePos 													:= Q_BasePos	:= FeedBasePos;
Done 														:= FALSE;
Busy 														:= True;
END_METHOD

METHOD PUBLIC WorkPos : BOOL //Return = Done
ToBasePos 													:= Q_BasePos 		:= FALSE;
ToWorkPos													:= TRUE;
Q_WorkPos	 												:= FeedWorkPos AND (NOT Options.7 OR NOT I_WorkPos);
WorkPos														:= Done 				:= I_WorkPos;
Busy														:= NOT Done;
END_METHOD

END_FUNCTION_BLOCK

// ---- POUs/Actuators/FreqConv/EcFcCom.TcPOU
{attribute 'no_check'}
FUNCTION_BLOCK EcFcCom (* SEW *)
VAR_INPUT
	StartLeft												:	BOOL := FALSE;
	StartRight												:	BOOL := FALSE;
	InAck													:	BOOL := TRUE;
	Contactor												:	BOOL := FALSE;(* if available *)
	Enable													:	BOOL := FALSE;
	FeedLeft												:	BOOL := TRUE;
	FeedRight												:	BOOL := TRUE;
	Velo													: 	LREAL := 0.0; (* speed of rotation *)
	Ramp													:	LREAL := 1.0;
	ProtSwitchOK											: 	FUSE;
	FuseBreakOK												: 	FUSE;
END_VAR                     							
VAR_OUTPUT                  							
	Ready													:	BOOL;
	Warning													:	BOOL;
	Busy													:	BOOL;
	Error													:	BOOL;
{attribute 'displaymode':='binary'}
	Status													:	BYTE; (* for HMI *)
{attribute 'displaymode':='binary'}
	UnitStatus												:	BYTE; (* devicestatus
																	0x0 not ready
																	0x1 controller locked
																	0x2 not enabled
																	0x3 standstill current acitve, not enabled
																	0x4 enabled
																	0x8 default factory settings active *)
	ErrorCode												:	BYTE; (* see also SEW-documentary *)
	Statuswort1										AT  %I* : 	INT;
	ActVelo													: 	LREAL;
	ActCurrent										AT  %I* : 	INT;
END_VAR                 							
VAR (* IO Internal *)   							
	_Steuerwort1									AT  %Q* : 	INT;
	_SetVeloDigit									AT  %Q* : 	INT;
	_Rampe											AT  %Q* :	INT;
                        							
	_Contactor 										AT  %Q* :	BOOL;
	_ActVeloDigit									AT  %I* : 	INT; (* rpm *)
END_VAR                 								
VAR                     	
	AckIntern												:	BOOL;
END_VAR

(* Com SEW MovitracB over Ethercat Gateway 		V2.0	*)
(********************************************************)

(* Protection Switch *****************************************)
	IF InAck 
	THEN 
		Ack(); 
	END_IF
	
	ProtSwitchOK(
		Force	:= ,
		Invert	:= ,
		InAck 	:= AckIntern,
		Q		=> ,
		Event 	=> ,
		INPUT 	=> );
	
	FuseBreakOK(InAck := AckIntern); (* same parameter like ProtSwitch *)

(* Contactor ********************************************************)
	_Contactor 												:= Contactor AND ProtSwitchOK.Q AND FuseBreakOK.Q;

(* Statuswort Auswerten *********************************)
	(*EndstufeFRG											:= Statuswort1.0; *)
	Ready													:= Statuswort1.1 AND _Contactor;
	Warning													:= Statuswort1.5 AND Ready ;
	Error													:= Statuswort1.5 AND NOT Ready AND _Contactor ;
	(*EndlLinksAktiv 										:= Statuswort1.6; *)
	(*EndlLinksAktiv 										:= Statuswort1.7; *)
                        									
	ActVelo													:= INT_TO_LREAL(_ActVeloDigit) * 0.2;
	Busy													:= Ready AND _Steuerwort1.2 AND ActVelo > 5.0;
                        	
(* Auswertung HighByte Statuswort 1 ********************)
	(* Init *)
	UnitStatus 												:= ErrorCode := 0;

IF _Contactor THEN
	IF NOT Statuswort1.5 THEN
		UnitStatus.0 										:= Statuswort1.8;
		UnitStatus.1 										:= Statuswort1.9;
		UnitStatus.2 										:= Statuswort1.10;
		UnitStatus.3										:= Statuswort1.11;
		UnitStatus.4 										:= Statuswort1.12;
		UnitStatus.5 										:= Statuswort1.13;
		UnitStatus.6 										:= Statuswort1.14;
		UnitStatus.7 										:= Statuswort1.15;
	ELSE                									
		ErrorCode.0 										:= Statuswort1.8;
		ErrorCode.1 										:= Statuswort1.9;
		ErrorCode.2 										:= Statuswort1.10;
		ErrorCode.3											:= Statuswort1.11;
		ErrorCode.4 										:= Statuswort1.12;
		ErrorCode.5 										:= Statuswort1.13;
		ErrorCode.6 										:= Statuswort1.14;
		ErrorCode.7 										:= Statuswort1.15;
	END_IF
END_IF

(* write contorlword 1  *********************************)
	_Steuerwort1.0 											:= FALSE; (* controller locked=1/0=enabled *)
	_Steuerwort1.1 											:= Enable AND _Contactor; (* controller enabled=1/0=rapid stop *)
	_Steuerwort1.2 											:= FeedLeft AND StartLeft AND NOT StartRight
																OR FeedRight AND StartRight AND NOT StartLeft; (* enable start FU *)
	_Steuerwort1.6 											:= AckIntern;
	_Steuerwort1.8 											:= NOT StartRight AND StartLeft; (* rotation direction 0=right/1=left *)
                        									
(* setvalue **************************************)
	IF 	StartRight 
		AND NOT StartLeft 
		AND FeedRight 
	THEN
		_SetVeloDigit 										:= LREAL_TO_INT(Velo) * 5; (* 5 Digit = 1 rpm *)
	ELSIF StartLeft 
		AND NOT StartRight 
		AND FeedLeft 
	THEN
		_SetVeloDigit 										:= (LREAL_TO_INT(Velo) * 5 ) * -1; (* 5 Digit = 1 rpm *)
	ELSE
		_SetVeloDigit 										:= 0;
	END_IF

(* set ramp ******************************************)
	_Rampe	 												:= LREAL_TO_INT(Ramp);

(* Ack FALSE **********************************************)
	AckIntern												:= FALSE;
	
(* HmiStatus **************************************************)
	Status.0 												:= _Steuerwort1.2 AND _Steuerwort1.8 ; //counter-clockwise rotation
	Status.1 												:= _Steuerwort1.2 AND NOT  _Steuerwort1.8; //clockwise rotation
	Status.2 												:= FALSE;
	Status.3												:= FALSE;
	Status.4 												:= FeedLeft;
	Status.5 												:= FeedRight;
	Status.7 												:= Ready;
	Status.7 												:= Error;
	                    									

(**************************************************************)

METHOD PUBLIC Ack
VAR_INPUT
END_VAR
AckIntern 													:= _Steuerwort1.6 := TRUE;
END_METHOD

METHOD PUBLIC SetContactorOFF
VAR_INPUT
END_VAR
_Contactor 													:= Contactor :=FALSE;
SETDISABLE();												
SETSTOP();
END_METHOD

METHOD PUBLIC SetContactorON
VAR_INPUT
END_VAR
_Contactor 													:= Contactor := ProtSwitchOK.Q AND FuseBreakOK.Q ;
END_METHOD

METHOD PUBLIC SetDisable
VAR_INPUT
END_VAR
Enable 														:= FALSE;
_Steuerwort1.1 												:= FALSE;
END_METHOD

METHOD PUBLIC SetEnable
VAR_INPUT
END_VAR
Enable 														:= TRUE;
_Steuerwort1.1 												:= _Contactor; (* FRGRegler=1/0=Schnellstopp *)
END_METHOD

METHOD PUBLIC SetStartLeft
VAR_INPUT
END_VAR
StartRight 													:= FALSE;
StartLeft													:= TRUE;
                									
_Steuerwort1.2 												:= FeedLeft AND StartLeft; (* FRG Start FU *)
_Steuerwort1.8 												:= StartRight AND NOT StartLeft; (* Drehrichtung 0=Rechts/1=Links *)
END_METHOD

METHOD PUBLIC SetStartRight
VAR_INPUT
END_VAR
StartRight 													:= TRUE;
StartLeft													:= FALSE;
                											
_Steuerwort1.2 												:= FeedRight AND StartRight AND NOT StartLeft; (* FRG Start FU *)
_Steuerwort1.8 												:= StartRight AND NOT StartLeft; (* Drehrichtung 0=Rechts/1=Links *)
END_METHOD

METHOD PUBLIC SetStop
VAR_INPUT
END_VAR
StartRight 													:= FALSE;
StartLeft													:= FALSE;
_Steuerwort1.2 												:= FALSE;
END_METHOD

END_FUNCTION_BLOCK

// ---- POUs/Actuators/FreqConv/IOFcCom.TcPOU
{attribute 'no_check'}
FUNCTION_BLOCK IOFcCom (* Frequence Converter IO Com *)
VAR_INPUT
	StartLeft												:	BOOL := FALSE;
	StartRight												:	BOOL := FALSE;
	InAck													:	BOOL := TRUE;
	Velo													:	LREAL := 0.0;
	VeloMin													:	LREAL := 0.0;
	VeloMax													:	LREAL := 100.0;
	FeedLeft												:	BOOL := TRUE;
	FeedRight												:	BOOL := TRUE;
	Contactor												:	BOOL;(* wenn vorhanden *)
	PT_DelBreak												:	TIME := T#1000MS;
	PT_DelEnable											:	TIME := T#1000MS;
	ProtSwitchOK											: 	FUSE;
	FuseBreakOK												: 	FUSE;
END_VAR         								
VAR_OUTPUT      								
	Ready											AT  %I* : 	BOOL := TRUE;
	Error											AT  %I* : 	BOOL := FALSE;
	Busy													:	BOOL;
{attribute 'displaymode':='binary'}
	Status													:	BYTE;
END_VAR
VAR (* IO Internal *)
	_SetValue										AT  %Q* : 	INT;
	_Reset											AT  %Q* :	BOOL;
	_Enable											AT  %Q* :	BOOL;
	_StartLeft										AT  %Q* :	BOOL;
	_StartRight										AT  %Q* :	BOOL;
	_Break											AT  %Q* :	BOOL; (* if available *)
	_Contactor										AT  %Q* :	BOOL;
END_VAR             								
VAR                 								
	TOF_Break												:	TOF;
	TOF_Enable												:	TOF;
	AckIntern												:	BOOL;
	BreakOpenIntern											:	BOOL;
END_VAR

(* Com FC IO 										 		V1.3	*)
(********************************************************************)

(* Protection Switch ************************************************)
	IF InAck 
	THEN 
		Ack(); 
	END_IF

	ProtSwitchOK(
		Force	:= ,
		Invert	:= ,
		InAck 	:= AckIntern,
		Q		=> ,
		Event 	=> ,
		INPUT 	=> );
		
	FuseBreakOK(InAck := AckIntern); (* same parameter like ProtSwitch *)

(* Contactor ********************************************************)
	_Contactor 												:= Contactor AND ProtSwitchOK.Q AND FuseBreakOK.Q;
	
(* Start ********************************************)
	IF 	StartRight 
		AND NOT StartLeft
	THEN
		SetStartRight();
	ELSIF StartLeft 
		AND NOT StartRight
	THEN
		SetStartLeft();
	ELSE
		 SetStop();
   END_IF

(* Enable ****************************************************)
	TOF_Enable(	IN := _SetValue <> 0,
					PT := PT_DelEnable);

	_Enable 												:= TOF_Enable.Q AND Ready AND _Break;

(* setvalue standardization *********************************)
	IF VeloMax > VeloMin THEN
		IF Velo >= VeloMax THEN
			_SetValue 										:= 32767;
		ELSIF Velo < VeloMin                				
		THEN                                				
			_SetValue 										:= 0;
		ELSE                                				
			_SetValue										:=LREAL_TO_INT ((32767.0 / (VeloMax - VeloMin)) * (Velo - VeloMin));
		END_IF                              				
	ELSE                                    				
		_SetValue 											:= 0;
	END_IF                                  				

(* setvalue **************************************)
	IF _StartLeft THEN
		_SetValue 											:= ABS(_SetValue) * -1;
	ELSIF _StartRight THEN              			
		_SetValue 											:= ABS(_SetValue);
	ELSE                                			
		_SetValue 											:= 0;
	END_IF                              	

(* HmiStatus **************************************************)
	Status.0 												:= _StartLeft AND Ready AND _Contactor;
	Status.1 												:= _StartRight AND Ready AND _Contactor;
	Status.2 												:= FALSE;
	Status.3 												:= _Break;
	Status.4 												:= FeedLeft ;
	Status.5 												:= FeedRight;
	Status.6 												:= Ready;
	Status.7 												:= Error;
	                                				
(* Status ***********************************************************)
	Busy 													:= TOF_Enable.Q AND TOF_Break.ET <= MAX(T#500MS,TOF_Break.PT) - T#500MS ;
	
(* Break ************************************************************)
	TOF_Break(	IN := _SetValue <> 0,
					PT := PT_DelBreak);

	IF _SetValue <> 0 
	THEN 
		BreakOpenIntern := FALSE; 
	END_IF

	_Break 													:= TOF_Break.Q AND Ready OR BreakOpenIntern;

(* Reset ***********************************************************)
	_Reset 													:= InAck OR AckIntern;
	AckIntern 												:= FALSE;

(**************************************************************)

METHOD PUBLIC Ack
VAR_INPUT
END_VAR
_Reset 														:= AckIntern 	:= TRUE;
END_METHOD

METHOD PUBLIC SetBreakClose
VAR_INPUT
END_VAR
BreakOpenIntern 											:= FALSE;
END_METHOD

METHOD PUBLIC SetBreakOpen
VAR_INPUT
END_VAR
BreakOpenIntern 							:= TRUE;
END_METHOD

METHOD PUBLIC SetContactorOFF
VAR_INPUT
END_VAR
Contactor 													:= FALSE;
SetStop();
END_METHOD

METHOD PUBLIC SetContactorON
VAR_INPUT
END_VAR
Contactor 													:= TRUE;
END_METHOD

METHOD PUBLIC SetStartLeft
VAR_INPUT
END_VAR
StartLeft 													:= TRUE; 
StartRight 													:= FALSE;
_StartLeft 													:= _Contactor AND Ready AND NOT Error AND FeedLeft;
END_METHOD

METHOD PUBLIC SetStartRight
VAR_INPUT
END_VAR
StartLeft 													:= FALSE; 
StartRight 													:= TRUE;
_StartRight 												:= _Contactor AND Ready AND NOT Error and FeedRight;
END_METHOD

METHOD PUBLIC SetStop
VAR_INPUT
END_VAR
StartLeft 													:= StartRight := _StartLeft := _StartRight := FALSE;
END_METHOD

END_FUNCTION_BLOCK

// ---- POUs/Actuators/Motor/IOMotorStarDelta.TcPOU
{attribute 'no_check'}
FUNCTION_BLOCK IOMotorStarDelta
VAR_INPUT
	InAck													:	BOOL := TRUE;
	StartRight												:	BOOL := FALSE;
	FeedRight												:	BOOL := TRUE;
	PT_RestartDel											:	TIME := T#0S;
	PT_Delta												: 	TIME := T#5S;
	ProtSwitchOK											: 	FUSE;
	ProtSwitchOK2											: 	FUSE;
END_VAR                 						
VAR_OUTPUT              						
	Busy													:	BOOL;
	Error													:	BOOL;
	Status													:	BYTE;
	RestartDelActive										:	BOOL;
	ET_RestartDel											: 	TIME;	(* waiting-time of start interlock *)
END_VAR                 						
VAR                     						
	TON_StarDelta											:	TON;
	TP_RestartDel											:	TP;
	_StarContactor									AT %Q* 	: 	BOOL;
	_DeltaContactor									AT %Q* 	: 	BOOL;
	_MainContactor									AT %Q* 	: 	BOOL;
END_VAR

(* Start Delta Motor IO	 				 	V1.1	*)
(****************************************************)

(* Protection Switch *****************************************)
	IF InAck 
	THEN 
		Ack(); 
	END_IF

	ProtSwitchOK(
		Force	:= ,
		Invert	:= ,
		InAck 	:= FALSE,
		Q		=> ,
		Event	=> ,
		INPUT 	=> );

	ProtSwitchOK2(InAck 	:= FALSE);
	
(* Start ****************************************************)
	IF StartRight THEN
		_MainContactor 										:= 	NOT TP_RestartDel.Q
																AND ProtSwitchOK.Q 
																AND ProtSwitchOK2.Q	
																AND FeedRight;
                       										
		_StarContactor 										:= 	_MainContactor
																AND NOT TON_StarDelta.Q
																AND NOT _DeltaContactor;

		_DeltaContactor 									:= 	_MainContactor
																AND TON_StarDelta.Q;

		TP_RestartDel();
	ELSE
		TP_RestartDel(IN := _MainContactor , PT := PT_RestartDel);
		_MainContactor 										:= FALSE;
		_DeltaContactor 									:= FALSE;
		_StarContactor 										:= FALSE;
	END_IF

(* Timer *****************************************************)
	TON_StarDelta( IN := _MainContactor, PT := PT_Delta);

(* Status ***********************************************************)
	Busy	 												:= _MainContactor;
	Error													:= NOT ProtSwitchOK.Q OR NOT ProtSwitchOK2.Q; 
	RestartDelActive										:= TP_RestartDel.Q;
	
	IF TP_RestartDel.ET > T#0MS 
	THEN
		ET_RestartDel		:= TP_RestartDel.PT - TP_RestartDel.ET;
	ELSE
		ET_RestartDel		:= t#0ms;
	END_IF
	
(* HmiStatus **************************************************)
	Status.0												 := NOT _MainContactor;
	Status.1												 := _MainContactor;
	Status.2												 := _DeltaContactor;
	Status.3												 := RestartDelActive;
	Status.4												 := FALSE;
	Status.5												 := FeedRight;
	Status.6												 := NOT Error AND NOT RestartDelActive;
	Status.7												 := Error;

(*********************************************************************)

METHOD PUBLIC Ack
VAR_INPUT
END_VAR
ProtSwitchOK(InAck := TRUE);
ProtSwitchOK2(InAck := TRUE);
END_METHOD

METHOD PUBLIC Reset
VAR_INPUT
END_VAR
Ack();
SetStop();
END_METHOD

METHOD PUBLIC ResetRestartTmr
VAR_INPUT
END_VAR
MEMSET(ADR(TP_RestartDel),0,SIZEOF(TP_RestartDel));
END_METHOD

METHOD PUBLIC SetStartRight
VAR_INPUT
END_VAR
StartRight 													:= TRUE;
END_METHOD

METHOD PUBLIC SetStop
VAR_INPUT
END_VAR
StartRight 													:= FALSE;
_MainContactor 												:= FALSE;
_DeltaContactor 											:= FALSE;
_StarContactor 												:= FALSE;
END_METHOD

END_FUNCTION_BLOCK

// ---- POUs/Actuators/SensorikAbblasen.TcPOU
{attribute 'no_check'}
FUNCTION_BLOCK SensorikAbblasen
VAR_INPUT
	Enable													:	BOOL;
	StartManual												:	BOOL;
	Abblasintervall											:	TIME := T#5M;
	Abblasdauer												:	TIME := t#4s;
	Abblastakt												:	TIME := t#500ms;
END_VAR                 									
VAR_OUTPUT              									
	Aktiv													:	BOOL;
	Q_DWORD													:	DWORD := 0;
END_VAR                 									
VAR                     									
	state													:	INT := 0;
	i														:	SINT ;
	TON_Abblasintervall										:	TON;
	TON_Abblasdauer 										: 	TON;
	TOF_Abblastakt 											:	TOF;
END_VAR

(* Abblastaktgenerator					*)
(***************************************)

(* Intervalzeit ***********************************************************************)
IF Enable 
THEN
	CASE state OF
	0:
		TON_Abblasintervall(IN := FALSE);
		state 												:= 10;
		i 													:= -1;

	1:
		Aktiv := FALSE;
		TON_Abblasintervall(IN := Abblasintervall <> t#0ms , PT := Abblasintervall);
		IF TON_Abblasintervall.Q
			OR StartManual
		THEN
			TON_Abblasintervall(IN := FALSE);
			
			state 											:= 10;
			Aktiv 											:= TRUE;
			i 												:= -1;
		END_IF

	10:
		i := i + 1;
		IF i > 31 THEN
			state 											:= 1;
		ELSE
			TON_Abblasdauer(IN := FALSE);
			TOF_Abblastakt(IN := FALSE);
			
			Q_DWORD 										:= 0;
			state 											:= 11;
		END_IF                  							

